# B&R Automation Studio project NAEUL004C00R13L518F00 (part 38)

#### Act_Alarm.st
```iecst
(** 2019-03-25 **)
ACTION Act_Alarm:

	//Error
	IF EDGEPOS(eStatus = Error) THEN

		tyAlmData.sProgNm		:= p_sProgNm;
		tyAlmData.udiCode		:= udiStatus;
		tyAlmData.eSeverity		:= AlmSeverityError;
		tyAlmData.udiRunTime	:= tyAlmData.udiRunTime + 1;
		tyAlmData.bAlm			:= TRUE;
		tyAlmData.udiModuleNum  := udiModuleNum;
		g_sUsrMgmtProgNm		:= p_sProgNm;

		//Get Error Message
		IF tyAlmData.udiCode < 10000 OR tyAlmData.udiCode > 10099 THEN
			tyAlmData.sAlmMsg	:= 'Unknown';
			tyAlmData.sRcyMsg	:= 'Unknown';
		ELSE
			tyAlmData.sAlmMsg	:= a_tyAlmText[tyAlmData.udiCode].sAlmText;
			tyAlmData.sRcyMsg	:= a_tyAlmText[tyAlmData.udiCode].sRcyText;
		END_IF

		sStatTxt	:= tyAlmData.sAlmMsg;

	ELSIF bRstErr AND (tyAlmData.udiCode <> 0) THEN

		tyAlmData.udiCode	:= 0;
		tyAlmData.eSeverity	:= AlmSeverityNA;
		tyAlmData.sAlmMsg	:= '';
		tyAlmData.sRcyMsg	:= '';
		tyAlmData.bAlm			:= FALSE;
		sStatTxt	:= a_sStatText[eStat];

	END_IF

END_ACTION
```

### Package Logical/OvenInfo - cmp

### OvenInfo.typ - Do Not Change!!!
```iecst
(*2018-12-13*)
(**)
(*Action*)

TYPE
	eOvenInfoAction :
		(
		OvenInfoActIdle,
		OvenInfoActSetBrdInOven,
		OvenInfoActSetOvenAllow,
		OvenInfoActRstOvenAllow
		);
	tyOvenInfo : 	STRUCT
		In : tyOvenInfoIn1;
		Out : tyOvenInfoOut1;
	END_STRUCT;
	tyOvenInfoIn1 : 	STRUCT
		eAct : eOvenInfoAction; (*Hardware Info's Action*)
		bPrep : BOOL := TRUE; (*Project Preparation*)
		bEn : BOOL := TRUE; (*Enable*)
		bDis : BOOL := FALSE; (*Disable*)
		bPrepExtdd : BOOL;
		bEnExtdd : BOOL;
		bDisExtdd : BOOL;
		bManual : BOOL;
		diBffrMtySlt : DINT;
		diAddBffr : DINT;
		diSetBrdInOven : DINT;
		bCntUp : BOOL;
		bCntDown : BOOL;
		bLinkOpsStatusRun : BOOL;
		eLinkOpsTravLifPosGo : REFERENCE TO eTravLifULPos;
		usiLinkProdRcpCurrRcpMcMod : REFERENCE TO USINT;
		diMinBffr : REFERENCE TO DINT;
		bBGRun : BOOL;
		BrdPerSlt : DINT;
		bLinkConvHvBrd : BOOL;
	END_STRUCT;
	tyOvenInfoOut1 : 	STRUCT
		eStat : eOvenInfoAction := OvenInfoActIdle; (*Hardware Info's State*)
		eStatus : eFBStatus := Idle; (*Hardware Info's Status*)
		sStatTxt : STRING[200] := ''; (*Hardware Info's State in Text*)
		tyAlmData : tyAlmDat; (*Alarm Data*)
		bOvenAllow : BOOL;
		diBrdInOven : DINT;
	END_STRUCT;
END_TYPE
```

### OvenInfo.var - Change By Project
```iecst
VAR
	g_tyOvenInfoA : tyOvenInfoOut1;
	g_tyOvenInfoB : tyOvenInfoOut1;
END_VAR
```

### Program Logical/OvenInfo/OvenInfoA (IEC, version 1.00.0) - 1.00.0 - NtOvenInfo v5.00.0

#### Init.st - Change By Project
```iecst
(** 2019-03-25 **)
PROGRAM _INIT

	(* Always Change If Project Change *)

	//Pass Address To Global Address For External Use
	//Action, State & Status
	p_OvenInfoAStat		:= ADR(eStat);
	p_OvenInfoAStatus	:= ADR(eStatus);
	p_OvenInfoAStatTxt	:= ADR(sStatTxt);

	//Alarm

	//Output
	p_OvenInfoAOvenAllow	:= ADR(bOvenAllow);
	p_OvenInfoABrdInOven	:= ADR(diBrdInOven);

	(* Always Change If Project Change *)

END_PROGRAM
```

#### Act_InitGlobal.st - Change By Project
```iecst
(** 2019-04-04 **)
ACTION Act_InitGlobal:

	(* Always Change If Project Change *)

	//Pass Data To Link
	p_bLinkOpsStatusRun ACCESS p_OpsStatusRun;
//	p_usiLinkProdRcpCurrRcpMcMod ACCESS p_ProdRcpCurrRcp2McMod;
	p_eLinkOpsTravLifPosGo ACCESS p_OpsTravLifULPosGo;
	p_eLinkConvStat ACCESS p_PshrConvStat;
	p_bLinkConvHvBrd ACCESS p_PshrConvHvBrd;

	//Pass Data To Internal Use
	p_eAct ACCESS p_UIOvenInfoAAct;
	p_bPrep ACCESS p_NtParamOvenInfoPrep;
	p_bEn ACCESS p_McParamOvenEn;
	p_bPrepExtdd ACCESS p_NtParamOvenInfoExtdPrep;
	p_bEnExtdd ACCESS p_McParamExtdOvenEn;
	p_bManual ACCESS p_UIMnlMod;
	p_diBffrMtySlt ACCESS p_BufferMagABffrMtySlt;
	//p_diMinBffr ACCESS p_ProdRcpCurrRcp2MinReqFreeBffr;
	p_diAddBffr ACCESS p_McParamOvenMaxBffr;
	p_diSetBrdInOven ACCESS p_UIOvenInfoSetBrdInOvenA;
	p_bCntUp ACCESS p_DIOvenInfeedSigA;
	p_bNtSettingsLoadDone ACCESS p_StartupNtSettingsLoadDone;

	p_bNtParamAutoRcpPrep ACCESS p_NtParamAutoRcpPrep;
	p_bMcParamAutoRcpDis  ACCESS p_McParamAutoRcpDisable;
	p_eNtParamAutoRcpPrecededBy ACCESS p_NtParamAutoRcpPrecededBy;
	(* Always Change If Project Change *)

END_ACTION
```

#### InputRef_Link.var - Change By Project
```iecst
(*2019-04-04*)
(**)
(*External*)
VAR
	p_bLinkOpsStatusRun : REFERENCE TO BOOL;
	p_usiLinkProdRcpCurrRcpMcMod : REFERENCE TO USINT;
	p_eLinkOpsTravLifPosGo : REFERENCE TO eTravLifULPos;
	p_eLinkConvStat : REFERENCE TO eConvAction;
	p_bLinkConvHvBrd : REFERENCE TO BOOL;
END_VAR
```

#### Act_LinkAction.st - Change By Project
```iecst
(** 2019-04-04 **)
ACTION Act_LinkAction:

	IF EDGENEG(p_bManual) THEN
		p_eAct	:= OvenInfoActIdle;
	END_IF

END_ACTION
```

#### Act_Link.st - Change By Project
```iecst
(** 2019-03-29 **)
ACTION Act_Link:
	IF g_tyNtParamCurr.bAutoRcpPrep AND NOT(g_tyMcParamCurr.bAutoRcpDisable) THEN //AutoRcp Ignored Follower
		tylocalOvenInfoA.In.usiLinkProdRcpCurrRcpMcMod ACCESS p_ProdRcpCurrRcp0McMod;
		tylocalOvenInfoA.In.diMinBffr ACCESS p_ProdRcpCurrRcp0MinReqFreeBffr;
	ELSE
		tylocalOvenInfoA.In.usiLinkProdRcpCurrRcpMcMod ACCESS p_ProdRcpCurrRcp1McMod;
		tylocalOvenInfoA.In.diMinBffr ACCESS p_ProdRcpCurrRcp2MinReqFreeBffr;
	END_IF

	tylocalOvenInfoA.In.bBGRun	:= tylocalOvenInfoA.In.bLinkOpsStatusRun
					AND (tylocalOvenInfoA.In.usiLinkProdRcpCurrRcpMcMod = ULModUnloadFrontLnA OR tylocalOvenInfoA.In.usiLinkProdRcpCurrRcpMcMod = ULModRejFrontLnA
					OR tylocalOvenInfoA.In.usiLinkProdRcpCurrRcpMcMod = ULModRejFrontLnARev OR tylocalOvenInfoA.In.usiLinkProdRcpCurrRcpMcMod = ULModUnloadDualLnAB
					OR tylocalOvenInfoA.In.usiLinkProdRcpCurrRcpMcMod = ULModRejDualLnA OR tylocalOvenInfoA.In.usiLinkProdRcpCurrRcpMcMod = ULModRejDualLnB);

	tylocalOvenInfoA.In.bCntDown 	:= tylocalOvenInfoA.In.eLinkOpsTravLifPosGo = TravLifULPosUS1 AND tylocalOvenInfoA.In.eLinkConvStat = ConvActEnt AND tylocalOvenInfoA.In.bLinkConvHvBrd = TRUE;

END_ACTION
```

#### Cyclic.st - Do Not Change!!!
```iecst
(** 2019-03-29 **)
PROGRAM _CYCLIC

	IF bInitialDone = FALSE THEN
		IF g_tyStartUp.bNtSettingsLoadDone = TRUE  THEN
			bInitialDone	:= TRUE;
			Act_Initial;
		END_IF

	ELSE

		IF (tylocalOvenInfoA.In.bPrep = TRUE) AND (tylocalOvenInfoA.In.bEn = TRUE) AND (tylocalOvenInfoA.In.bDis = FALSE) THEN
			Act_InputConfig;
			Act_Link;
			Act_Main;
			Act_OutputConfig;
		ELSE
			Act_Main_Disable;

			IF tylocalOvenInfoA.Out.eStat <> OvenInfoActIdle THEN
				tylocalOvenInfoA.Out.eStatus	:= Done;
			ELSE
				tylocalOvenInfoA.Out.eStatus	:= Idle;
			END_IF
		END_IF

	END_IF

END_PROGRAM
```

#### Act_Initial.st - Do Not Change!!!
```iecst
(** 2019-01-03 **)
ACTION Act_Initial:

	//Initial
	sStatTxt	:= a_sStatText[eStat];

	fbStd(bEn := FALSE);
	fbExtdd(bEn := FALSE);

END_ACTION
```

#### Act_Main.st - Do Not Change!!!
```iecst
(** 2019-01-10 **)
ACTION Act_Main:

	IF EDGENEG(g_tyUIOut.bManualMod) THEN
		tylocalOvenInfoA.In.eAct	:= OvenInfoActIdle;
	END_IF
	//Set tylocalOvenInfoA.In.eAct
	IF tylocalOvenInfoA.Out.eStatus = Idle OR tylocalOvenInfoA.Out.eStatus = Busy OR tylocalOvenInfoA.Out.eStatus = Done THEN
		tylocalOvenInfoA.Out.eStat	:= tylocalOvenInfoA.In.eAct;
	END_IF

	IF tylocalOvenInfoA.Out.eStatOld <> tylocalOvenInfoA.Out.eStat THEN
		tylocalOvenInfoA.Out.sStatTxt	:= a_sStatText[tylocalOvenInfoA.Out.eStat];

		tylocalOvenInfoA.Out.eStatOld	:= tylocalOvenInfoA.Out.eStat;

		tylocalOvenInfoA.Out.eStatus		:= Busy;
	END_IF

	//Main
	CASE tylocalOvenInfoA.Out.eStat OF

		OvenInfoActIdle:
			tylocalOvenInfoA.Out.eStatus	:= Idle;

		OvenInfoActSetBrdInOven:
			IF tylocalOvenInfoA.Out.eStatus = Idle OR tylocalOvenInfoA.Out.eStatus = Busy THEN

				tylocalOvenInfoA.Out.diBrdInOven	:= tylocalOvenInfoA.In.diSetBrdInOven;
				tylocalOvenInfoA.Out.eStatus		:= Done;

			END_IF

		OvenInfoActSetOvenAllow:
			IF tylocalOvenInfoA.Out.eStatus = Idle OR tylocalOvenInfoA.Out.eStatus = Busy THEN

				tylocalOvenInfoA.Out.bOvenAllow	:= TRUE;
				tylocalOvenInfoA.Out.eStatus		:= Done;

			END_IF

		OvenInfoActRstOvenAllow:
			IF tylocalOvenInfoA.Out.eStatus = Idle OR tylocalOvenInfoA.Out.eStatus = Busy THEN

				tylocalOvenInfoA.Out.bOvenAllow	:= FALSE;
				tylocalOvenInfoA.Out.eStatus		:= Done;

			END_IF

	END_CASE

	IF tylocalOvenInfoA.In.bManual = TRUE THEN
		fbStd(bEn := FALSE);
		fbExtdd(bEn := FALSE);

	ELSIF tylocalOvenInfoA.In.bBGRun = FALSE THEN
		fbStd(bEn := FALSE);
		fbExtdd(bEn := FALSE);

		tylocalOvenInfoA.Out.bOvenAllow	:= FALSE;

	ELSIF (tylocalOvenInfoA.In.bPrepExtdd = TRUE) AND (tylocalOvenInfoA.In.bEnExtdd = TRUE) AND (tylocalOvenInfoA.In.bDisExtdd = FALSE) THEN

		fbStd(bEn := FALSE);

		IF EDGEPOS(tylocalOvenInfoA.In.bCntUp) THEN
			tylocalOvenInfoA.Out.diBrdInOven	:= tylocalOvenInfoA.Out.diBrdInOven + 1;
		END_IF

		IF EDGEPOS(tylocalOvenInfoA.In.bCntDown) THEN
			tylocalOvenInfoA.Out.diBrdInOven	:= tylocalOvenInfoA.Out.diBrdInOven - 1;
		END_IF

		IF tylocalOvenInfoA.Out.diBrdInOven < 0 THEN
			tylocalOvenInfoA.Out.diBrdInOven	:= 0;
		END_IF

		fbExtdd.diAddBffr		:= tylocalOvenInfoA.In.diAddBffr;
		fbExtdd.diBffrMtySlt	:= tylocalOvenInfoA.In.diBffrMtySlt;
		fbExtdd.diBrdInOven		:= tylocalOvenInfoA.Out.diBrdInOven;
		fbExtdd.diBrdPerSlt		:= tylocalOvenInfoA.In.diBrdPerSlt;
		fbExtdd(bEn := TRUE);
		tylocalOvenInfoA.Out.bOvenAllow	:= fbExtdd.bOvenAllow;

	ELSE

		fbExtdd(bEn := FALSE);

		fbStd.diBffrMtySlt		:= tylocalOvenInfoA.In.diBffrMtySlt;
		fbStd.diMinBffrMtySlt	:= tylocalOvenInfoA.In.diMinBffr;
		fbStd(bEn := TRUE);
		tylocalOvenInfoA.Out.bOvenAllow	:= fbStd.bOvenAllow;

	END_IF

END_ACTION
```

#### Act_Main_Disable.st - Do Not Change!!!
```iecst
(** 2019-01-24 **)
ACTION Act_Main_Disable:

	tylocalOvenInfoA.Out.bOvenAllow	:= TRUE;

END_ACTION
```

#### InputRef.var - Do Not Change!!!
```iecst
(*2019-04-04*)
(**)
(*General*)
VAR
	p_eAct : REFERENCE TO eOvenInfoAction;
END_VAR
(**)
VAR
	p_bPrep : REFERENCE TO BOOL;
	p_bEn : REFERENCE TO BOOL;
	p_bDis : REFERENCE TO BOOL;
	p_bPrepExtdd : REFERENCE TO BOOL;
	p_bEnExtdd : REFERENCE TO BOOL;
	p_bDisExtdd : REFERENCE TO BOOL;
END_VAR
(**)
(*Configuration*)
VAR
	p_bBGRun : REFERENCE TO BOOL;
	p_bManual : REFERENCE TO BOOL;
	p_diBffrMtySlt : REFERENCE TO DINT;
	p_diMinBffr : REFERENCE TO DINT;
	p_diAddBffr : REFERENCE TO DINT;
	p_diBrdPerSlt : REFERENCE TO DINT;
	p_bCntUp : REFERENCE TO BOOL;
	p_bCntDown : REFERENCE TO BOOL;
	p_diSetBrdInOven : REFERENCE TO DINT;
	p_bNtSettingsLoadDone : REFERENCE TO BOOL;
END_VAR
(*AutoRcp*)
VAR
	p_bNtParamAutoRcpPrep : REFERENCE TO BOOL;
	p_bMcParamAutoRcpDis : REFERENCE TO BOOL;
	p_eNtParamAutoRcpPrecededBy : REFERENCE TO eAutoRcpPreceded;
END_VAR
```

#### Local.var - Do Not Change!!!
```iecst
(*2019-04-30*)
(**)
VAR
	tylocalOvenInfoA : tyOvenInfo;
	a_sStatText : ARRAY[0..50] OF STRING[200] := ['Idling','Setting Board In Oven Value','Turning On Oven Allow Output','Turning Off Oven Allow Output',47('')];
END_VAR
(**)
(*Local Alarm*)
(**)
(*Local Output*)
VAR
	bOvenAllow : BOOL;
END_VAR
VAR RETAIN
	diBrdInOven : DINT;
END_VAR
(**)
(*Local Input*)
VAR
	bPrep : BOOL := TRUE;
	bEn : BOOL := TRUE;
	bDis : BOOL := FALSE;
	bPrepExtdd : BOOL := TRUE;
	bEnExtdd : BOOL := TRUE;
	bDisExtdd : BOOL := FALSE;
	bBGRun : BOOL := FALSE;
	bManual : BOOL := FALSE;
	diBffrMtySlt : DINT;
	diMinBffr : DINT;
	diAddBffr : DINT;
	diBrdPerSlt : DINT := 1;
	bCntUp : BOOL;
	bCntDown : BOOL;
	diSetBrdInOven : DINT;
	bNtSettingsLoadDone : BOOL := TRUE;
END_VAR
(**)
(*Local*)
VAR
	bInitDone : BOOL;
	bInitialDone : BOOL;
	fbStd : fbOvenInfoStd;
	fbExtdd : fbOvenInfoExtdd;
	eStatOld : eOvenInfoAction := OvenInfoActIdle;
END_VAR
```

#### Act_InputConfig.st - not listed in the package file held
```iecst
ACTION Act_InputConfig:

	//Pass Data To Link
	tylocalOvenInfoA.In.bLinkOpsStatusRun :=  g_tyOps.bStatusRun;
	//	p_usiLinkProdRcpCurrRcpMcMod ACCESS p_ProdRcpCurrRcp2McMod;
	tylocalOvenInfoA.In.eLinkOpsTravLifPosGo ACCESS p_OpsTravLifULPosGo;
	tylocalOvenInfoA.In.eLinkConvStat := g_tyPshrConv.eStat;
	tylocalOvenInfoA.In.bLinkConvHvBrd := g_tyPshrConv.bHvBrd;

	//Pass Data To Internal Use
	tylocalOvenInfoA.In.eAct := g_tyUIOut.eOvenInfoAAct;
	tylocalOvenInfoA.In.bPrep := g_tyNtParam.bOvenInfoPrep;
	tylocalOvenInfoA.In.bEn := g_tyMcParamCurr.bOvenEn;
	tylocalOvenInfoA.In.bPrepExtdd := g_tyNtParam.bOvenInfoExtdPrep;
	tylocalOvenInfoA.In.bEnExtdd := g_tyMcParamCurr.bExtdOvenEn;
	tylocalOvenInfoA.In.bManual := g_tyUIOut.bMnlMod;
	tylocalOvenInfoA.In.diBffrMtySlt  := g_tyBufferMagA.diBffrMtySlt;
	//tylocalOvenInfoA.In.diMinBffr ACCESS p_ProdRcpCurrRcp2MinReqFreeBffr;
	tylocalOvenInfoA.In.diAddBffr := g_tyMcParamCurr.diOvenMaxBffr;
	tylocalOvenInfoA.In.diSetBrdInOven := g_tyUIOut.diOvenInfoSetBrdInOvenA;
	tylocalOvenInfoA.In.bCntUp := g_tyDInput.bOvenInfeedSigA;

	(* Always Change If Project Change *)

END_ACTION
```

#### Act_OutputConfig.st - not listed in the package file held
```iecst
ACTION Act_OutputConfig:

	g_tyOvenInfoA := tylocalOvenInfoA.Out;

END_ACTION
```

### Program Logical/OvenInfo/OvenInfoB (IEC) - 1.00.0 - NtOvenInfo v5.00.0

#### InputRef.var
```iecst
(*2019-04-04*)
(**)
(*General*)
VAR
	p_eAct : REFERENCE TO eOvenInfoAction;
END_VAR
(**)
VAR
	p_bPrep : REFERENCE TO BOOL;
	p_bEn : REFERENCE TO BOOL;
	p_bDis : REFERENCE TO BOOL;
	p_bPrepExtdd : REFERENCE TO BOOL;
	p_bEnExtdd : REFERENCE TO BOOL;
	p_bDisExtdd : REFERENCE TO BOOL;
END_VAR
(**)
(*Configuration*)
VAR
	p_bBGRun : REFERENCE TO BOOL;
	p_bManual : REFERENCE TO BOOL;
	p_diBffrMtySlt : REFERENCE TO DINT;
	p_diMinBffr : REFERENCE TO DINT;
	p_diAddBffr : REFERENCE TO DINT;
	p_diBrdPerSlt : REFERENCE TO DINT;
	p_bCntUp : REFERENCE TO BOOL;
	p_bCntDown : REFERENCE TO BOOL;
	p_diSetBrdInOven : REFERENCE TO DINT;
	p_bNtSettingsLoadDone : REFERENCE TO BOOL;
END_VAR
(*AutoRcp*)
VAR
	p_bNtParamAutoRcpPrep : REFERENCE TO BOOL;
	p_bMcParamAutoRcpDis1 : REFERENCE TO BOOL;
	p_eNtParamAutoRcpPrecededBy : REFERENCE TO eAutoRcpPreceded;
	p_bMcParamAutoRcpDis : REFERENCE TO BOOL;
END_VAR
```

#### InputRef_Link.var
```iecst
(*2019-04-04*)
(**)
(*External Data*)
VAR
	p_bLinkNtParamPrepB : REFERENCE TO BOOL;
	p_bLinkNtParamOvenInfoPrep : REFERENCE TO BOOL;
	p_bLinkOpsStatusRun : REFERENCE TO BOOL;
	p_usiLinkProdRcpCurrRcpMcMod : REFERENCE TO USINT;
	p_eLinkOpsTravLifPosGo : REFERENCE TO eTravLifULPos;
	p_eLinkConvStat : REFERENCE TO eConvAction;
	p_bLinkConvHvBrd : REFERENCE TO BOOL;
END_VAR
```

#### Local.var
```iecst
(*2019-04-30*)
VAR
	tylocalOvenInfoB : tyOvenInfo;
	a_sStatText : ARRAY[0..50] OF STRING[200] := ['Idling','Setting Board In Oven Value','Turning On Oven Allow Output','Turning Off Oven Allow Output',47('')];
END_VAR
(**)
(*Local Alarm*)
(**)
(*Local Output*)
VAR
	bOvenAllow : BOOL;
END_VAR
VAR RETAIN
	diBrdInOven : DINT;
END_VAR
(**)
(*Local Input*)
VAR
	bPrep : BOOL := TRUE;
	bEn : BOOL := TRUE;
	bDis : BOOL := FALSE;
	bPrepExtdd : BOOL := TRUE;
	bEnExtdd : BOOL := TRUE;
	bDisExtdd : BOOL := FALSE;
	bBGRun : BOOL := FALSE;
	bManual : BOOL := FALSE;
	diBffrMtySlt : DINT;
	diMinBffr : DINT;
	diAddBffr : DINT;
	diBrdPerSlt : DINT := 1;
	bCntUp : BOOL;
	bCntDown : BOOL;
	diSetBrdInOven : DINT;
	bNtSettingsLoadDone : BOOL := TRUE;
END_VAR
(**)
(*Local*)
VAR
	bInitDone : BOOL;
	bInitialDone : BOOL;
	fbStd : fbOvenInfoStd;
	fbExtdd : fbOvenInfoExtdd;
	eStatOld : eOvenInfoAction := OvenInfoActIdle;
END_VAR
```

#### Act_Background.st
```iecst
(** 2019-05-15 **)
ACTION Act_Background:

	IF p_bManual = TRUE THEN
		fbStd(bEn := FALSE);
		fbExtdd(bEn := FALSE);

	ELSIF p_bBGRun = FALSE THEN
		fbStd(bEn := FALSE);
		fbExtdd(bEn := FALSE);

		bOvenAllow	:= FALSE;

	ELSIF (p_bPrepExtdd = TRUE) AND (p_bEnExtdd = TRUE) AND (p_bDisExtdd = FALSE) THEN

		fbStd(bEn := FALSE);

		IF EDGEPOS(p_bCntUp) THEN
			diBrdInOven	:= diBrdInOven + 1;
		END_IF

		IF EDGEPOS(p_bCntDown) THEN
			diBrdInOven	:= diBrdInOven - 1;
		END_IF

		IF diBrdInOven < 0 THEN
			diBrdInOven	:= 0;
		END_IF

		fbExtdd.diAddBffr		:= p_diAddBffr;
		fbExtdd.diBffrMtySlt	:= p_diBffrMtySlt;
		fbExtdd.diBrdInOven		:= diBrdInOven;
		fbExtdd.diBrdPerSlt		:= p_diBrdPerSlt;
		fbExtdd(bEn := TRUE);
		bOvenAllow	:= fbExtdd.bOvenAllow;

	ELSE

		fbExtdd(bEn := FALSE);

		fbStd.diBffrMtySlt		:= p_diBffrMtySlt;
		fbStd.diMinBffrMtySlt	:= p_diMinBffr;
		fbStd(bEn := TRUE);
		bOvenAllow	:= fbStd.bOvenAllow;

	END_IF

END_ACTION
```

#### Act_InitGlobal.st
```iecst
(** 2019-04-04 **)
ACTION Act_InitGlobal:

	(* Always Change If Project Change *)

	//Pass Data To Link
	p_bLinkNtParamPrepB ACCESS p_NtParamProjLaneBPrep;
	p_bLinkNtParamOvenInfoPrep ACCESS p_NtParamOvenInfoPrep;
	p_bLinkOpsStatusRun ACCESS p_OpsStatusRun;
//	p_usiLinkProdRcpCurrRcpMcMod ACCESS p_ProdRcpCurrRcp2McMod;
	p_eLinkOpsTravLifPosGo ACCESS p_OpsTravLifULPosGo;
	p_eLinkConvStat ACCESS p_PshrConvStat;
	p_bLinkConvHvBrd ACCESS p_PshrConvHvBrd;

	//Pass Data To Internal Use
	p_eAct ACCESS p_UIOvenInfoBAct;
	p_bEn ACCESS p_McParamOvenEn;
	p_bPrepExtdd ACCESS p_NtParamOvenInfoExtdPrep;
	p_bEnExtdd ACCESS p_McParamExtdOvenEn;
	p_bManual ACCESS p_UIMnlMod;
	p_diBffrMtySlt ACCESS p_BufferMagBBffrMtySlt;
//	p_diMinBffr ACCESS p_ProdRcpCurrRcp2MinReqFreeBffr;
	p_diAddBffr ACCESS p_McParamOvenMaxBffr;
	p_diSetBrdInOven ACCESS p_UIOvenInfoSetBrdInOvenB;
	p_bCntUp ACCESS p_DIOvenInfeedSigB;
	p_bNtSettingsLoadDone ACCESS p_StartupNtSettingsLoadDone;

	p_bNtParamAutoRcpPrep ACCESS p_NtParamAutoRcpPrep;
	p_bMcParamAutoRcpDis  ACCESS p_McParamAutoRcpDisable;
	p_eNtParamAutoRcpPrecededBy ACCESS p_NtParamAutoRcpPrecededBy;
	(* Always Change If Project Change *)

END_ACTION
```

#### Act_Initial.st
```iecst
(** 2019-01-03 **)
ACTION Act_Initial:

	//Initial
	tylocalOvenInfoA.Out.sStatTxt	:= a_sStatText[tylocalOvenInfoA.Out.eStat];

	fbStd(bEn := FALSE);
	fbExtdd(bEn := FALSE);

END_ACTION
```

#### Act_InitLocal.st
```iecst
(** 2019-04-04 **)
ACTION Act_InitLocal:

	//Input Reference Link To Local Variable
	p_eAct ACCESS ADR(eAct);
	p_bPrep ACCESS ADR(bPrep);
	p_bEn ACCESS ADR(bEn);
	p_bDis ACCESS ADR(bDis);
	p_bPrepExtdd ACCESS ADR(bPrepExtdd);
	p_bEnExtdd ACCESS ADR(bEnExtdd);
	p_bDisExtdd ACCESS ADR(bDisExtdd);
	p_bBGRun ACCESS ADR(bBGRun);
	p_bManual ACCESS ADR(bManual);
	p_diMinBffr ACCESS ADR(diMinBffr);
	p_diAddBffr ACCESS ADR(diAddBffr);
	p_diBffrMtySlt ACCESS ADR(diBffrMtySlt);
	p_diBrdPerSlt ACCESS ADR(diBrdPerSlt);
	p_bCntUp ACCESS ADR(bCntUp);
	p_bCntDown ACCESS ADR(bCntDown);
	p_diSetBrdInOven ACCESS ADR(diSetBrdInOven);
	p_bNtSettingsLoadDone ACCESS ADR(bNtSettingsLoadDone);

END_ACTION
```

#### Act_InputConfig.st
```iecst
ACTION Act_InputConfig:

	(* Always Change If Project Change *)

	//Pass Data To Link
	tylocalOvenInfoB.In.bLinkOpsStatusRun :=  g_tyOps.bStatusRun;
	//	p_usiLinkProdRcpCurrRcpMcMod ACCESS p_ProdRcpCurrRcp2McMod;
	tylocalOvenInfoB.In.eLinkOpsTravLifPosGo ACCESS p_OpsTravLifULPosGo;
	tylocalOvenInfoB.In.eLinkConvStat := g_tyPshrConv.eStat;
	tylocalOvenInfoB.In.bLinkConvHvBrd := g_tyPshrConv.bHvBrd;

	tylocalOvenInfoB.In.eAct := g_tyUIOut.eOvenInfoBAct;
	//tylocalOvenInfoB.In.bPrep := g_tyNtParam.bOvenInfoPrep;
	tylocalOvenInfoB.In.bEn := g_tyMcParamCurr.bOvenEn;
	tylocalOvenInfoB.In.bPrepExtdd := g_tyNtParam.bOvenInfoExtdPrep;
	tylocalOvenInfoB.In.bEnExtdd := g_tyMcParamCurr.bExtdOvenEn;
	tylocalOvenInfoB.In.bManual := g_tyUIOut.bMnlMod;
	tylocalOvenInfoB.In.diBffrMtySlt  := g_tyBufferMagB.diBffrMtySlt;
	//tylocalOvenInfoB.In.diMinBffr ACCESS p_ProdRcpCurrRcp2MinReqFreeBffr;
	tylocalOvenInfoB.In.diAddBffr := g_tyMcParamCurr.diOvenMaxBffr;
	tylocalOvenInfoB.In.diSetBrdInOven := g_tyUIOut.diOvenInfoSetBrdInOvenB;
	tylocalOvenInfoB.In.bCntUp := g_tyDInput.bOvenInfeedSigB;

	//Link bPrep, bEn & bDis
	tylocalOvenInfoB.In.bPrep	:= g_tyNtParamCurr.bOvenInfoPrep AND g_tyNtParamCurr.bProjLaneBPrep;

END_ACTION
```

#### Act_Link.st
```iecst
(** 2019-03-29 **)
ACTION Act_Link:

	IF g_tyNtParamCurr.bAutoRcpPrep AND NOT(g_tyMcParamCurr.bAutoRcpDisable) THEN //AutoRcp Ignored Follower
		tylocalOvenInfoB.In.usiLinkProdRcpCurrRcpMcMod ACCESS p_ProdRcpCurrRcp0McMod;
		tylocalOvenInfoB.In.diMinBffr ACCESS p_ProdRcpCurrRcp0MinReqFreeBffr;
	ELSE
		tylocalOvenInfoB.In.usiLinkProdRcpCurrRcpMcMod ACCESS p_ProdRcpCurrRcp1McMod;
		tylocalOvenInfoB.In.diMinBffr ACCESS p_ProdRcpCurrRcp2MinReqFreeBffr;
	END_IF

	tylocalOvenInfoB.In.bBGRun := 	tylocalOvenInfoB.In.bLinkOpsStatusRun
					AND (tylocalOvenInfoB.In.usiLinkProdRcpCurrRcpMcMod = ULModUnloadRearLnB OR tylocalOvenInfoB.In.usiLinkProdRcpCurrRcpMcMod = ULModRejRearLnB
					OR tylocalOvenInfoB.In.usiLinkProdRcpCurrRcpMcMod = ULModRejRearLnBRev OR tylocalOvenInfoB.In.usiLinkProdRcpCurrRcpMcMod = ULModUnloadDualLnAB
					OR tylocalOvenInfoB.In.usiLinkProdRcpCurrRcpMcMod = ULModRejDualLnA OR tylocalOvenInfoB.In.usiLinkProdRcpCurrRcpMcMod = ULModRejDualLnB);

	tylocalOvenInfoA.In.bCntDown	:= p_eLinkOpsTravLifPosGo = TravLifULPosUS2 AND p_eLinkConvStat = ConvActEnt AND p_bLinkConvHvBrd = TRUE;

END_ACTION
```

#### Act_LinkEn.st
```iecst
(** 2019-01-11 **)
ACTION Act_LinkEn:

	//Link bPrep, bEn & bDis
	p_bPrep	:= p_bLinkNtParamOvenInfoPrep AND p_bLinkNtParamPrepB;

END_ACTION
```

#### Act_Main.st
```iecst
(** 2019-01-10 **)
ACTION Act_Main:

	IF EDGENEG(g_tyUIOut.bManualMod) THEN
		tylocalOvenInfoB.In.eAct	:= OvenInfoActIdle;
	END_IF
	//Set tylocalOvenInfoB.In.eAct
	IF tylocalOvenInfoB.Out.eStatus = Idle OR tylocalOvenInfoB.Out.eStatus = Busy OR tylocalOvenInfoB.Out.eStatus = Done THEN
		tylocalOvenInfoB.Out.eStat	:= tylocalOvenInfoB.In.eAct;
	END_IF

	IF tylocalOvenInfoB.Out.eStatOld <> tylocalOvenInfoB.Out.eStat THEN
		tylocalOvenInfoB.Out.sStatTxt	:= a_sStatText[tylocalOvenInfoB.Out.eStat];

		tylocalOvenInfoB.Out.eStatOld	:= tylocalOvenInfoB.Out.eStat;

		tylocalOvenInfoB.Out.eStatus		:= Busy;
	END_IF

	//Main
	CASE tylocalOvenInfoB.Out.eStat OF

		OvenInfoActIdle:
			tylocalOvenInfoB.Out.eStatus	:= Idle;

		OvenInfoActSetBrdInOven:
			IF tylocalOvenInfoB.Out.eStatus = Idle OR tylocalOvenInfoB.Out.eStatus = Busy THEN

				tylocalOvenInfoB.Out.diBrdInOven	:= tylocalOvenInfoB.In.diSetBrdInOven;
				tylocalOvenInfoB.Out.eStatus		:= Done;

			END_IF

		OvenInfoActSetOvenAllow:
			IF tylocalOvenInfoB.Out.eStatus = Idle OR tylocalOvenInfoB.Out.eStatus = Busy THEN

				tylocalOvenInfoB.Out.bOvenAllow	:= TRUE;
				tylocalOvenInfoB.Out.eStatus		:= Done;

			END_IF

		OvenInfoActRstOvenAllow:
			IF tylocalOvenInfoB.Out.eStatus = Idle OR tylocalOvenInfoB.Out.eStatus = Busy THEN

				tylocalOvenInfoB.Out.bOvenAllow	:= FALSE;
				tylocalOvenInfoB.Out.eStatus		:= Done;

			END_IF

	END_CASE

	IF tylocalOvenInfoB.In.bManual = TRUE THEN
		fbStd(bEn := FALSE);
		fbExtdd(bEn := FALSE);

	ELSIF tylocalOvenInfoB.In.bBGRun = FALSE THEN
		fbStd(bEn := FALSE);
		fbExtdd(bEn := FALSE);

		tylocalOvenInfoB.Out.bOvenAllow	:= FALSE;

	ELSIF (tylocalOvenInfoB.In.bPrepExtdd = TRUE) AND (tylocalOvenInfoB.In.bEnExtdd = TRUE) AND (tylocalOvenInfoB.In.bDisExtdd = FALSE) THEN

		fbStd(bEn := FALSE);

		IF EDGEPOS(tylocalOvenInfoB.In.bCntUp) THEN
			tylocalOvenInfoB.Out.diBrdInOven	:= tylocalOvenInfoB.Out.diBrdInOven + 1;
		END_IF

		IF EDGEPOS(tylocalOvenInfoB.In.bCntDown) THEN
			tylocalOvenInfoB.Out.diBrdInOven	:= tylocalOvenInfoB.Out.diBrdInOven - 1;
		END_IF

		IF tylocalOvenInfoB.Out.diBrdInOven < 0 THEN
			tylocalOvenInfoB.Out.diBrdInOven	:= 0;
		END_IF

		fbExtdd.diAddBffr		:= tylocalOvenInfoB.In.diAddBffr;
		fbExtdd.diBffrMtySlt	:= tylocalOvenInfoB.In.diBffrMtySlt;
		fbExtdd.Out.diBrdInOven		:= tylocalOvenInfoB.Out.diBrdInOven;
		fbExtdd.diBrdPerSlt		:= tylocalOvenInfoB.In.diBrdPerSlt;
		fbExtdd(bEn := TRUE);
		tylocalOvenInfoB.Out.bOvenAllow	:= fbExtdd.Out.bOvenAllow;

	ELSE

		fbExtdd(bEn := FALSE);

		fbStd.diBffrMtySlt		:= tylocalOvenInfoB.In.diBffrMtySlt;
		fbStd.diMinBffrMtySlt	:= tylocalOvenInfoB.In.diMinBffr;
		fbStd(bEn := TRUE);
		tylocalOvenInfoB.Out.bOvenAllow	:= fbStd.Out.bOvenAllow;

	END_IF

END_ACTION
```

#### Act_Main_Disable.st
```iecst
(** 2019-01-24 **)
ACTION Act_Main_Disable:

	tylocalOvenInfoB.Out.bOvenAllow= TRUE;

END_ACTION
```

#### Act_OutputConfig.st
```iecst
ACTION Act_OutputConfig:

	g_tyOvenInfoB := tylocalOvenInfoB.Out;

END_ACTION
```

#### Cyclic.st
```iecst
(** 2019-03-29 **)
PROGRAM _CYCLIC

	IF bInitialDone = FALSE THEN
		IF g_tyStartUp.bNtSettingsLoadDone = TRUE  THEN
			bInitialDone	:= TRUE;
			Act_Initial;
		END_IF

	ELSE

		IF (tylocalOvenInfoB.In.bPrep = TRUE) AND (tylocalOvenInfoB.In.bEn = TRUE) AND (tylocalOvenInfoB.In.bDis = FALSE) THEN
			Act_InputConfig;
			Act_Link;
			Act_Main;
			Act_OutputConfig;
		ELSE
			Act_Main_Disable;

			IF tylocalOvenInfoB.Out.eStat <> OvenInfoActIdle THEN
				tylocalOvenInfoB.Out.eStatus	:= Done;
			ELSE
				tylocalOvenInfoB.Out.eStatus	:= Idle;
			END_IF
		END_IF

	END_IF

END_PROGRAM
```

#### Init.st
```iecst
(** 2019-03-25 **)
PROGRAM _INIT

	(* Always Change If Project Change *)

	//Pass Address To Global Address For External Use
	//Action, State & Status
	p_OvenInfoBStat		:= ADR(eStat);
	p_OvenInfoBStatus	:= ADR(eStatus);
	p_OvenInfoBStatTxt	:= ADR(sStatTxt);

	//Alarm

	//Output
	p_OvenInfoBOvenAllow	:= ADR(bOvenAllow);
	p_OvenInfoBBrdInOven	:= ADR(diBrdInOven);

	(* Always Change If Project Change *)

END_PROGRAM
```

### OvenInfoA.var - not listed in the package file held
```iecst
(*2019-03-25*)
(**)
(*Action & State & Status*)
VAR
	p_OvenInfoAStat : UDINT;
	p_OvenInfoAStatus : UDINT;
	p_OvenInfoAStatTxt : UDINT;
END_VAR
(**)
(*Alarm*)
(**)
(*Output*)
VAR
	p_OvenInfoAOvenAllow : UDINT;
	p_OvenInfoABrdInOven : UDINT;
END_VAR
```

### OvenInfoB.var - not listed in the package file held
```iecst
(*2019-03-25*)
(**)
(*Action & State & Status*)
VAR
	p_OvenInfoBStat : UDINT;
	p_OvenInfoBStatus : UDINT;
	p_OvenInfoBStatTxt : UDINT;
END_VAR
(**)
(*Alarm*)
(**)
(*Output*)
VAR
	p_OvenInfoBOvenAllow : UDINT;
	p_OvenInfoBBrdInOven : UDINT;
END_VAR
```

### Buffer.typ - Do Not Change!!!
```iecst
(*2019-02-18*)
(**)
(*Action*)

TYPE
	eBufferAction :
		(
		BufferActIdle,
		BufferActCreateDir,
		BufferActGetRetainBffr,
		BufferActSetFull,
		BufferActSetMty,
		BufferActLoad,
		BufferActLoadSltChk,
		BufferActUnload,
		BufferActUnloadSltChk,
		BufferActUnloadCoolChk,
		BufferActUnloadSltChkCoolChk,
		BufferActNxtLoad,
		BufferActNxtLoadGd,
		BufferActNxtLoadBad,
		BufferActNxtUnload,
		BufferActNxtUnloadGd,
		BufferActNxtUnloadBad,
		BufferActChkCoolTm,
		BufferActChkCoolBrdAny,
		BufferActChkCoolBrdGd,
		BufferActChkCoolBrdBad,
		BufferActRstBffr,
		BufferActSetCoolFan,
		BufferActRstCoolFan,
		BufferActBGStartBffrSetFull,
		BufferActBGStartBffrSetMty,
		BufferActBGStopBffrSet,
		BufferActBGStartUpdtSen,
		BufferActBGStopUpdtSen,
		BufferActBGStartUpdtDisplay,
		BufferActBGStopUpdtDisplay,
		BufferActBGStartCoolFan,
		BufferActBGStopCoolFan
		);
	tyBuffer1 : 	STRUCT
		In : tyBufferIn1;
		Out : tyBufferOut1;
	END_STRUCT;
	tyBufferIn1 : 	STRUCT
		eAct : eBufferAction; (*Hardware Info's Action*)
		udiRstErr : UDINT;
		sFileName : STRING[80];
		bManual : BOOL;
		dtCurrDT : DATE_AND_TIME;
		diMinSlt : DINT;
		diMaxSlt : DINT;
		diPitch : DINT;
		diSltCap : DINT;
		diBffrTtlSlt : DINT;
		diCoolTm : DINT;
		diSltToSltInUM : DINT;
		diLifterBtmPosInUM : DINT;
		diLifterCurrPosInUM : DINT;
		bAscending : BOOL;
		bFIFO : BOOL;
		bGdBrdIn : BOOL;
		bGdBrdReq : BOOL;
		bNxtLoadSeq : BOOL;
		a_bSkip : ARRAY[1..c_diBffrSize]OF BOOL;
		diCoolFanOffDlyTm : DINT;
		bMagPresentSensor : BOOL;
		bPrepCoolFan : BOOL;
		bCoolFanTm : BOOL;
		tyBufferStat : tyBffrStat;
		sBffrNm : STRING[15];
		sProdNm : STRING[15];
		sBarcode1 : STRING[80];
		sBarcode2 : STRING[80];
		sCurrRcpNm : STRING[15];
		sProgNm : STRING[15];
		bNtSettingsLoadDone : BOOL;
		bNtParamAutoRcpPrep : BOOL;
		bMcParamAutoRcpDis : BOOL;
		bOpsMagConvULRlsMagAllw : BOOL;
		eNtParamCustomerReq : eCustomer;
		tyResponseFromMES : tyStatPlatformFromMES;
		diLinkSltToSltDist : REFERENCE TO DINT;
		bLinkMcParamProdSelTopToBtm : REFERENCE TO BOOL;
		bLinkPresentSen1 : BOOL;
		bLinkPresentSen2 : BOOL;
		bLinkOpsTravLifULExitBrd : REFERENCE TO BOOL;
	END_STRUCT;
	tyBufferOut1 : 	STRUCT
		eStat : eBufferAction := BufferActIdle; (*Hardware Info's State*)
		eStatus : eFBStatus := Idle; (*Hardware Info's Status*)
		sStatTxt : STRING[200] := ''; (*Hardware Info's State in Text*)
		tyAlmData : tyAlmDat; (*Alarm Data*)
		diNxtLoadSlt : DINT;
		diNxtUnloadSlt : DINT;
		diCoolBrdAny : DINT;
		diCoolBrdGd : DINT;
		diCoolBrdBad : DINT;
		bCoolNotRdy : BOOL;
		tyBuffer : tyBffr;
		tyDispBuffer : tyDispBffr;
		tyBufferStat : tyBffrStat;
		tyBoardUnloadStat : tyBrdUnloadStat;
		bCoolFanCtrl : BOOL;
		bParamDiff : BOOL;
		bMagRemoved : BOOL;
		bFIFOOld : BOOL;
		bMagPresent : BOOL;
		dtMagPresentTm : DATE_AND_TIME;
		diCurrSlt : DINT;
	END_STRUCT;
END_TYPE

(* *)

TYPE
	tyBufferMag : 	STRUCT
		In : tyBufferMagIn1;
		Out : tyBufferMagOut1;
	END_STRUCT;
	tyBufferMagIn1 : 	STRUCT
		eAct : eBufferAction; (*Hardware Info's Action*)
		udiRstErr : UDINT;
		bOpsStatusRun : BOOL;
		bBufferMagPresent1 : BOOL;
		bBufferMagPresent2 : BOOL;
		bBufferMagPresent3 : BOOL;
		bDIMagPresentSen1 : BOOL;
		bDIMagPresentSen2 : BOOL;
		bDIMagPresentSen3 : BOOL;
		tyBufferStat1 : tyBffrStat;
		tyBufferStat2 : tyBffrStat;
		tyBufferStat3 : tyBffrStat;
		bNtParamAutoRcpPrep : BOOL;
		bMcParamAutoRcpDis : BOOL;
		eNtParamMag : eULMag;
		bPrep : BOOL;
		bEn : BOOL;
		bDis : BOOL;
		usiProRcpProdSelMcMod : REFERENCE TO USINT;
	END_STRUCT;
	tyBufferMagOut1 : 	STRUCT
		eStat : eBufferAction := BufferActIdle; (*Hardware Info's State*)
		eStatus : eFBStatus := Idle; (*Hardware Info's Status*)
		sStatTxt : STRING[200] := ''; (*Hardware Info's State in Text*)
		tyAlmData : tyAlmDat; (*Alarm Data*)
		diBffrMtySlt : DINT;
	END_STRUCT;
END_TYPE
```

### Buffer.var - Change By Project
```iecst
VAR
	g_tyBuffer1 : tyBufferOut1;
	g_tyBuffer2 : tyBufferOut1;
	g_tyBuffer3 : tyBufferOut1;
	g_tyBufferMagA : tyBufferMagOut1;
	g_tyBufferMagB : tyBufferMagOut1;
END_VAR
```

### Program Logical/Buffer/Buffer1 (IEC) - 1.00.0 - NtBuffer v5.00.0 , NtFileIO v5.00.0

#### InputRef.var
```iecst
(*2019-07-03*)
(**)
(*General*)
VAR
	p_eAct : REFERENCE TO eBufferAction;
	p_udiRstErr : REFERENCE TO UDINT;
END_VAR
(**)
(*Configuration*)
VAR
	p_sFileName : REFERENCE TO STRING[80];
	p_bManual : REFERENCE TO BOOL;
	p_dtCurrDT : REFERENCE TO DATE_AND_TIME;
	p_diMinSlt : REFERENCE TO DINT;
	p_diMaxSlt : REFERENCE TO DINT;
	p_diPitch : REFERENCE TO DINT;
	p_diSltCap : REFERENCE TO DINT;
	p_diBffrTtlSlt : REFERENCE TO DINT;
	p_diCoolTm : REFERENCE TO DINT;
	p_diSltToSltInUM : REFERENCE TO DINT;
	p_diLifterBtmPosInUM : REFERENCE TO DINT;
	p_diLifterCurrPosInUM : REFERENCE TO DINT;
	p_bAscending : REFERENCE TO BOOL;
	p_bFIFO : REFERENCE TO BOOL;
	p_bGdBrdIn : REFERENCE TO BOOL;
	p_bGdBrdReq : REFERENCE TO BOOL;
	p_bNxtLoadSeq : REFERENCE TO BOOL;
	pa_bSkip : REFERENCE TO ARRAY[1..c_diBffrSize] OF BOOL;
	p_diCoolFanOffDlyTm : REFERENCE TO DINT;
	p_bMagPresentSensor : REFERENCE TO BOOL;
	p_bPrepCoolFan : REFERENCE TO BOOL;
	p_bCoolFanTm : REFERENCE TO BOOL;
	p_tyBuffer : REFERENCE TO tyBffr;
	p_tyDispBuffer : REFERENCE TO tyDispBffr;
	p_tyBufferStat : REFERENCE TO tyBffrStat;
	p_sBffrNm : REFERENCE TO STRING[15];
	p_sProdNm : REFERENCE TO STRING[15];
	p_sBarcode1 : REFERENCE TO STRING[80];
	p_sBarcode2 : REFERENCE TO STRING[80];
	p_sCurrRcpNm : REFERENCE TO STRING[15];
	p_sProgNm : REFERENCE TO STRING[15];
	p_bNtSettingsLoadDone : REFERENCE TO BOOL;
	p_bNtParamAutoRcpPrep : REFERENCE TO BOOL;
	p_bMcParamAutoRcpDis : REFERENCE TO BOOL;
	p_bOpsMagConvULRlsMagAllw : REFERENCE TO BOOL;
	p_eNtParamCustomerReq : REFERENCE TO eCustomer;
	p_tyResponseFromMES : REFERENCE TO tyStatPlatformFromMES;
	p_bNtParamAutoRcpF1ArbitraryType : REFERENCE TO BOOL;
END_VAR
```

#### InputRef_Link.var
```iecst
(*2019-04-09*)
(**)
(*External*)
VAR
	p_bLinkStartupRun : REFERENCE TO BOOL;
	p_bLinkNtParamProjMagConvPrep : REFERENCE TO BOOL;
	p_eLinkOpsMagULBufferAct : REFERENCE TO eBufferAction;
	p_eLinkOpsMagConvULBufferAct : REFERENCE TO eBufferAction;
	p_eLinkUIBufferAct : REFERENCE TO eBufferAction;
	p_bLinkOpsMagStepBffrLoad : REFERENCE TO BOOL;
END_VAR
(**)
VAR
	p_diLinkSltToSltDist : REFERENCE TO DINT;
	p_bLinkMcParamProdSelTopToBtm : REFERENCE TO BOOL;
	p_bLinkPresentSen1 : REFERENCE TO BOOL;
	p_bLinkPresentSen2 : REFERENCE TO BOOL;
	p_bLinkProjLifterMagPlatform : REFERENCE TO BOOL;
	p_eLinkOpsLifMagULBufferAct : REFERENCE TO eBufferAction;
	p_bLinkOpsTravLifULExitBrd : REFERENCE TO BOOL;
END_VAR
```

#### Local.var
```iecst
(*2019-06-07*)
(**)
(*Local Action, State & Status*)
VAR
	tylocalBuffer : tyBuffer1;
	eAct : eBufferAction;
	udiStatus : UDINT := 0;
	a_sStatText : ARRAY[0..50] OF STRING[200] := ['Idling','Creating Directory','Getting Retained Buffer Data','Setting Buffer Full','Setting Buffer Empty','Loading Board','Loading Board With Slot Check','Unloading Board','Unloading Board With Slot Check','Unloading Board With Cooling Time Check','Unloading Board With Slot Check And Cooling Time Check','Getting Next Load Board Slot Number','Getting Next Load Good Board Slot Number','Getting Next Load Bad Board Slot Number','Getting Next Unload Board Slot Number','Getting Next Unload Good Board Slot Number','Getting Next Unload Bad Board Slot Number','Checking Cooling Time','Checking Cooling Board','Checking Cooling Good Board','Checking Cooling Bad Board','Resetting Buffer','Turning On Cooling Fan','Turning Off Cooling Fan','Background Starting Buffer Set Full','Background Starting Buffer Set Empty','Background Stopping Buffer Set','Background Starting Update Sensor','Background Stopping Update Sensor','Background Starting Update Display','Background Stopping Update Display','Background Starting Cooling Fan','Background Stopping Cooling Fan',18('')];
END_VAR
(**)
(*Local Alarm*)
VAR
	tyAlmData : tyAlmDat;
	a_tyAlmText : ARRAY[10000..10099] OF tyAlmTxt := [(sAlmText:='Create User Directory Error',sRcyText:='An Error Occurred While Attempting To Create User Directory. Please Contact Nutek For A Possible Solution'),(sAlmText:='Create Retain Directory Error',sRcyText:='An Error Occurred While Attempting To Create Retain Directory. Please Contact Nutek For A Possible Solution'),(sAlmText:='File Open Error While Reading Retain File',sRcyText:='An Error Was Encountered While Trying To Open File. Please Contact Nutek For A Possible Solution.'),(sAlmText:='File Read Error While Reading Retain File',sRcyText:='An Error Was Encountered While Trying To Read File. Please Contact Nutek For A Possible Solution.'),(sAlmText:='File Close Error While Reading Retain File',sRcyText:='An Error Was Encountered While Trying To Close File. Please Contact Nutek For A Possible Solution.'),(sAlmText:='File Open Error While Setting Full Buffer',sRcyText:='An Error Was Encountered While Trying To Open File. Please Contact Nutek For A Possible Solution.'),(sAlmText:='File Create Error While Setting Full Buffer',sRcyText:='An Error Was Encountered While Trying To Create File. Please Contact Nutek For A Possible Solution.'),(sAlmText:='File Write Error While Setting Full Buffer',sRcyText:='An Error Was Encountered While Trying To Write File. Please Contact Nutek For A Possible Solution.'),(sAlmText:='File Close Error While Setting Full Buffer',sRcyText:='An Error Was Encountered While Trying To Close File. Please Contact Nutek For A Possible Solution.'),(sAlmText:='File Open Error While Setting Empty Buffer',sRcyText:='An Error Was Encountered While Trying To Open File. Please Contact Nutek For A Possible Solution.'),(sAlmText:='File Create Error While Setting Empty Buffer',sRcyText:='An Error Was Encountered While Trying To Create File. Please Contact Nutek For A Possible Solution.'),(sAlmText:='File Write Error While Setting Empty Buffer',sRcyText:='An Error Was Encountered While Trying To Write File. Please Contact Nutek For A Possible Solution.'),(sAlmText:='File Close Error While Setting Empty Buffer',sRcyText:='An Error Was Encountered While Trying To Close File. Please Contact Nutek For A Possible Solution.'),(sAlmText:='File Open Error While Loading Info To Buffer',sRcyText:='An Error Was Encountered While Trying To Open File. Please Contact Nutek For A Possible Solution.'),(sAlmText:='File Create Error While Loading Info To Buffer',sRcyText:='An Error Was Encountered While Trying To Create File. Please Contact Nutek For A Possible Solution.'),(sAlmText:='File Write Error While Loading Info To Buffer',sRcyText:='An Error Was Encountered While Trying To Write File. Please Contact Nutek For A Possible Solution.'),(sAlmText:='File Close Error While Loading Info To Buffer',sRcyText:='An Error Was Encountered While Trying To Close File. Please Contact Nutek For A Possible Solution.'),(sAlmText:='Wrong Slot Number To Load',sRcyText:='Invalid Slot to Load The Board.'),(sAlmText:='File Open Error While Loading Info To Buffer With Slot Check',sRcyText:='An Error Was Encountered While Trying To Open File. Please Contact Nutek For A Possible Solution.'),(sAlmText:='File Create Error While Loading Info To Buffer With Slot Check',sRcyText:='An Error Was Encountered While Trying To Create File. Please Contact Nutek For A Possible Solution.'),(sAlmText:='File Write Error While Loading Info To Buffer With Slot Check',sRcyText:='An Error Was Encountered While Trying To Write File. Please Contact Nutek For A Possible Solution.'),(sAlmText:='File Close Error While Loading Info To Buffer With Slot Check',sRcyText:='An Error Was Encountered While Trying To Close File. Please Contact Nutek For A Possible Solution.'),(sAlmText:='File Open Error While Unloading Info From Buffer',sRcyText:='An Error Was Encountered While Trying To Open File. Please Contact Nutek For A Possible Solution.'),(sAlmText:='File Create Error While Unloading Info From Buffer',sRcyText:='An Error Was Encountered While Trying To Create File. Please Contact Nutek For A Possible Solution.'),(sAlmText:='File Write Error While Unloading Info From Buffer',sRcyText:='An Error Was Encountered While Trying To Write File. Please Contact Nutek For A Possible Solution.'),(sAlmText:='File Close Error While Unloading Info From Buffer',sRcyText:='An Error Was Encountered While Trying To Close File. Please Contact Nutek For A Possible Solution.'),(sAlmText:='Wrong Slot Number To Unload',sRcyText:='Invalid Slot to Unload The Board.'),(sAlmText:='File Open Error While Unloading Info From Buffer With Slot Check',sRcyText:='An Error Was Encountered While Trying To Open File. Please Contact Nutek For A Possible Solution.'),(sAlmText:='File Create Error While Unloading Info From Buffer With Slot Check',sRcyText:='An Error Was Encountered While Trying To Create File. Please Contact Nutek For A Possible Solution.'),(sAlmText:='File Write Error While Unloading Info From Buffer With Slot Check',sRcyText:='An Error Was Encountered While Trying To Write File. Please Contact Nutek For A Possible Solution.'),(sAlmText:='File Close Error While Unloading Info From Buffer With Slot Check',sRcyText:='An Error Was Encountered While Trying To Close File. Please Contact Nutek For A Possible Solution.'),(sAlmText:='File Open Error While Unloading Info From Buffer With Cooling Time Check',sRcyText:='An Error Was Encountered While Trying To Open File. Please Contact Nutek For A Possible Solution.'),(sAlmText:='File Create Error While Unloading Info From Buffer With Cooling Time Check',sRcyText:='An Error Was Encountered While Trying To Create File. Please Contact Nutek For A Possible Solution.'),(sAlmText:='File Write Error While Unloading Info From Buffer With Cooling Time Check',sRcyText:='An Error Was Encountered While Trying To Write File. Please Contact Nutek For A Possible Solution.'),(sAlmText:='File Close Error While Unloading Info From Buffer With Cooling Time Check',sRcyText:='An Error Was Encountered While Trying To Close File. Please Contact Nutek For A Possible Solution.'),(sAlmText:='Wrong Slot Number To Unload With Cooling Time Check',sRcyText:='Invalid Slot to Unload The Board with Cooling Time Check.'),(sAlmText:='File Open Error While Unloading Info From Buffer With Slot Check And Cooling Time Check',sRcyText:='An Error Was Encountered While Trying To Open File. Please Contact Nutek For A Possible Solution.'),(sAlmText:='File Create Error While Unloading Info From Buffer With Slot Check And Cooling Time Check',sRcyText:='An Error Was Encountered While Trying To Create File. Please Contact Nutek For A Possible Solution.'),(sAlmText:='File Write Error While Unloading Info From Buffer With Slot Check And Cooling Time Check',sRcyText:='An Error Was Encountered While Trying To Write File. Please Contact Nutek For A Possible Solution.'),(sAlmText:='File Close Error While Unloading Info From Buffer With Slot Check And Cooling Time Check',sRcyText:='An Error Was Encountered While Trying To Close File. Please Contact Nutek For A Possible Solution.'),(sAlmText:='Directory Does Not Exist While Setting Full Buffer',sRcyText:='The Directory Does Not Exist. Please Contact Nutek For A Possible Solution.'),(sAlmText:='Directory Does Not Exist While Setting Empty Buffer',sRcyText:='The Directory Does Not Exist. Please Contact Nutek For A Possible Solution.'),(sAlmText:='Directory Does Not Exist While Loading Info To Buffer',sRcyText:='The Directory Does Not Exist. Please Contact Nutek For A Possible Solution.'),(sAlmText:='Directory Does Not Exist While Loading Info To Buffer With Slot Check',sRcyText:='The Directory Does Not Exist. Please Contact Nutek For A Possible Solution.'),(sAlmText:='Directory Does Not Exist While Unloading Info From Buffer',sRcyText:='The Directory Does Not Exist. Please Contact Nutek For A Possible Solution.'),(sAlmText:='Directory Does Not Exist While Unloading Info From Buffer With Slot Check',sRcyText:='The Directory Does Not Exist. Please Contact Nutek For A Possible Solution.'),(sAlmText:='Directory Does Not Exist While Unloading Info From Buffer With Cooling Time Check',sRcyText:='The Directory Does Not Exist. Please Contact Nutek For A Possible Solution.'),(sAlmText:='Directory Does Not Exist While Unloading Info From Buffer With Slot Check And Cooling Time Check',sRcyText:='The Directory Does Not Exist. Please Contact Nutek For A Possible Solution.'),(sAlmText:='Unloading Slot Is Skipped While Unloading Buffer',sRcyText:='Unload From Wrong Slot (Skip Slot).'),(sAlmText:='Unloading Slot Is Not For Board While Unloading Buffer',sRcyText:='Unload From Wrong Slot (Not For Board).'),(sAlmText:='Unloading Slot Board Is Not Available While Unloading Buffer',sRcyText:='Unload From Wrong Slot (Board Is Not Available).'),(sAlmText:='Unloading Last Sub Slot Is Not For Board While Unloading Buffer',sRcyText:='Unload From Wrong Slot (Last Sub Slot Is Not For Board).'),(sAlmText:='Unloading Last Sub Slot Has No Board While Unloading Buffer',sRcyText:='Unload From Wrong Slot (Last Sub Slot Has No Board).'),(sAlmText:='Board Quantity In Slot Is 0 While Unloading Buffer',sRcyText:='Unload From Wrong Slot (Board Quantity In Slot = 0).'),(sAlmText:='Board Capacity In Slot Is 0 While Unloading Buffer',sRcyText:='Unload From Wrong Slot (Board Capacity In Slot = 0).'),(sAlmText:='Unloading Slot Is Skipped While Unloading Buffer With Slot Check',sRcyText:='Unload From Wrong Slot (Skip Slot).'),(sAlmText:='Unloading Slot Is Not For Board While Unloading Buffer With Slot Check',sRcyText:='Unload From Wrong Slot (Not For Board).'),(sAlmText:='Unloading Slot Board Is Not available While Unloading Buffer With Slot Check',sRcyText:='Unload From Wrong Slot (Board Is Not Available).'),(sAlmText:='Unloading Last Sub Slot Is Not For Board While Unloading Buffer With Slot Check',sRcyText:='Unload From Wrong Slot (Last Sub Slot Is Not For Board).'),(sAlmText:='Unloading Last Sub Slot Has No Board While Unloading Buffer With Slot Check',sRcyText:='Unload From Wrong Slot (Last Sub Slot Has No Board).'),(sAlmText:='Board Quantity In Slot Is 0 While Unloading Buffer With Slot Check',sRcyText:='Unload From Wrong Slot (Board Quantity In Slot = 0).'),(sAlmText:='Board Capacity In Slot Is 0 While Unloading Buffer With Slot Check',sRcyText:='Unload From Wrong Slot (Board Capacity In Slot = 0).'),(sAlmText:='Unloading Slot Is Skipped While Unloading Buffer With Cool Check',sRcyText:='Unload From Wrong Slot (Skip Slot).'),(sAlmText:='Unloading Slot Is Not For Board While Unloading Buffer With Cool Check',sRcyText:='Unload From Wrong Slot (Not For Board).'),(sAlmText:='Unloading Slot Board Is Not available While Unloading Buffer With Cool Check',sRcyText:='Unload From Wrong Slot (Board Is Not Available).'),(sAlmText:='Unloading Last Sub Slot Is Not For Board While Unloading Buffer With Cool Check',sRcyText:='Unload From Wrong Slot (Last Sub Slot Is Not For Board).'),(sAlmText:='Unloading Last Sub Slot Has No Board While Unloading Buffer With Cool Check',sRcyText:='Unload From Wrong Slot (Last Sub Slot Has No Board).'),(sAlmText:='Board Quantity In Slot Is 0 While Unloading Buffer With Cool Check',sRcyText:='Unload From Wrong Slot (Board Quantity In Slot = 0).'),(sAlmText:='Board Capacity In Slot Is 0 While Unloading Buffer With Cool Check',sRcyText:='Unload From Wrong Slot (Board Capacity In Slot = 0).'),(sAlmText:='Unloading Slot Is Skipped While Unloading Buffer With Cool & Slot Check',sRcyText:='Unload From Wrong Slot (Skip Slot).'),(sAlmText:='Unloading Slot Is Not For Board While Unloading Buffer With Cool & Slot Check',sRcyText:='Unload From Wrong Slot (Not For Board).'),(sAlmText:='Unloading Slot Board Is Not available While Unloading Buffer With Cool & Slot Check',sRcyText:='Unload From Wrong Slot (Board Is Not Available).'),(sAlmText:='Unloading Last Sub Slot Is Not For Board While Unloading Buffer With Cool & Slot Check',sRcyText:='Unload From Wrong Slot (Last Sub Slot Is Not For Board).'),(sAlmText:='Unloading Last Sub Slot Has No Board While Unloading Buffer With Cool & Slot Check',sRcyText:='Unload From Wrong Slot (Last Sub Slot Has No Board).'),(sAlmText:='Board Quantity In Slot Is 0 While Unloading Buffer With Cool & Slot Check',sRcyText:='Unload From Wrong Slot (Board Quantity In Slot = 0).'),(sAlmText:='Board Capacity In Slot Is 0 While Unloading Buffer With Cool & Slot Check',sRcyText:='Unload From Wrong Slot (Board Capacity In Slot = 0).'),(sAlmText:='Loading Slot Is Not For Board',sRcyText:='Load To Wrong Slot (Not For Board).'),(sAlmText:='Loading Slot Is Full Of Board',sRcyText:='Load To Wrong Slot (Full With Board).'),(sAlmText:='Loading First Sub-Slot Is Not For Board',sRcyText:='Load To Wrong Slot (First Sub Slot Not For Board).'),(sAlmText:='Loading Last Sub-Slot Have Board, Which Mean Slot Is Full Of Board',sRcyText:='Load To Wrong Slot (Full With Board(Last Sub Slot Have Board)).'),(sAlmText:='Loading Last Sub-Slot Is Not For Board',sRcyText:='Load To Wrong Slot (Last Sub Slot Not For Board).'),(sAlmText:='Loading Slot Is Full Of Board',sRcyText:='Load To Wrong Slot (Full With Board).'),(sAlmText:='Loading Slot Is Skipped',sRcyText:='Load To Wrong Slot (Skip Slot).'),(sAlmText:='Existing Board Status Is Different With Loading Board Status',sRcyText:='Existing Board Status Is Different With Loading Buffer Status.'),(sAlmText:='Loading Slot Is Not For Board',sRcyText:='Load To Wrong Slot (Not For Board).'),(sAlmText:='Loading Slot Is Full Of Board',sRcyText:='Load To Wrong Slot (Full With Board).'),(sAlmText:='Loading First Sub-Slot Is Not For Board',sRcyText:='Load To Wrong Slot (First Sub Slot Not For Board).'),(sAlmText:='Loading Last Sub-Slot Have Board, Which Mean Slot Is Full Of Board',sRcyText:='Load To Wrong Slot (Full With Board(Last Sub Slot Have Board)).'),(sAlmText:='Loading Last Sub-Slot Is Not For Board',sRcyText:='Load To Wrong Slot (Last Sub Slot Not For Board).'),(sAlmText:='Loading Slot Is Full Of Board',sRcyText:='Load To Wrong Slot (Full With Board).'),(sAlmText:='Loading Slot Is Skipped',sRcyText:='Load To Wrong Slot (Skip Slot).'),(sAlmText:='Existing Board Status Is Different With Loading Board Status',sRcyText:='Existing Board Status Is Different With Loading Buffer Status.'),8((0))];
END_VAR
(**)
(**)
(**)
(*Local*)
VAR
	bRstErr : BOOL;
	udiRstErrOld : UDINT;
	bInitDone : BOOL;
	bInitialDone : BOOL;
	bUpdateSensor : BOOL;
	bBffrSetMty : BOOL;
	bBffrSetFull : BOOL;
	bUpdtDisplay : BOOL;
	usiStep : USINT;
	diCurrSlt : DINT;
	diExpectedSlt : DINT;
	bSetFull : BOOL;
	bSetMty : BOOL;
	bCoolFanRun : BOOL;
	tyBffrParameter : tyBffrParam;
	fbDirCreate1 : fbDirCreate;
	fbDirCreate2 : fbDirCreate;
	fbFileRead1 : fbFileFullRead;
	fbFileWrite1 : fbFileFullWrite;
	fbCoolFanOffDlyTm : TON;
	fbCoolFanOffChkTm : TON := (PT:=T#500ms);
	fbMagAbsentTm : TON := (PT:=T#5s);
	fbMagPresentTm : TON := (PT:=T#8s);
	eStatOld : eBufferAction := BufferActIdle;
	bMESTrigSetFull : BOOL;
	bFileNotFound : BOOL;
	bNewProduct : BOOL;
	bLastProductUnload : BOOL;
	bLastProductLeftInBffr : BOOL;
	udiModuleNum : UDINT := 2001;
END_VAR
```

#### Act_Background.st
```iecst
(** 2019-07-03 **)
ACTION Act_Background:

	fbMagPresentTm(IN := p_bMagPresentSensor);

	//Update Retain
	IF bUpdateSensor = TRUE THEN
		bMagPresent	:= fbMagPresentTm.Q;
	END_IF

	//Display Buffer
	IF bUpdtDisplay = TRUE THEN
		fDispBffrDescending(ADR(p_tyDispBuffer) , tyBffrParameter , p_tyBuffer , p_dtCurrDT , DINT_TO_TIME(p_diCoolTm) , 0 , 1 , 2);
	END_IF

	//Cooling Fan Control
	IF p_bManual = TRUE THEN
		;

	ELSIF bCoolFanRun = TRUE AND p_bPrepCoolFan = TRUE AND bCoolFanTm = TRUE THEN //Cooling Fan Control By Cooling Time

		fbCoolFanOffChkTm(IN := TRUE);

		IF fbCoolFanOffChkTm.Q = TRUE THEN
			IF fBffrChkCoolBrdAny(p_dtCurrDT, DINT_TO_TIME(p_diCoolTm), p_tyBuffer) = 0 THEN
				fbCoolFanOffDlyTm.IN	:= TRUE;
			ELSE
				fbCoolFanOffDlyTm.IN	:= FALSE;
				bCoolFanCtrl			:= TRUE;
			END_IF

			fbCoolFanOffChkTm(IN := FALSE);
		END_IF

		fbCoolFanOffDlyTm;

		IF fbCoolFanOffDlyTm.Q = TRUE THEN
			bCoolFanCtrl	:= FALSE;
		END_IF

	ELSIF bCoolFanRun = TRUE AND p_bPrepCoolFan = TRUE AND bCoolFanTm = FALSE THEN	//Cooling Fan Control By Buffer Empty
		fbCoolFanOffDlyTm(IN := p_tyBufferStat.bBffrMty);

		IF p_tyBufferStat.bBffrMty = FALSE THEN
			bCoolFanCtrl	:= TRUE;
		END_IF

		IF fbCoolFanOffDlyTm.Q = TRUE THEN
			bCoolFanCtrl	:= FALSE;
		END_IF

	ELSE

		bCoolFanCtrl	:= FALSE;

	END_IF

	//Set Buffer By Magazine Present
	IF bBffrSetFull = TRUE THEN
		IF p_bMagPresentSensor = TRUE AND fbMagAbsentTm.Q = TRUE THEN
			bSetFull		:= TRUE;
			dtMagPresentTm	:= p_dtCurrDT;
		END_IF

		IF bSetFull = TRUE  THEN
			p_eAct	:= BufferActSetFull;

			IF eStatus = Done AND eStat = BufferActSetFull THEN
				p_eAct		:= BufferActIdle;
				bSetFull	:= FALSE;
			ELSIF eStatus = Error THEN
				bSetFull	:= FALSE;
			END_IF
		END_IF

		fbMagAbsentTm(IN := NOT p_bMagPresentSensor);

	ELSIF bBffrSetMty = TRUE THEN
		IF p_bMagPresentSensor = TRUE AND fbMagAbsentTm.Q = TRUE THEN
			bSetMty			:= TRUE;
			dtMagPresentTm	:= p_dtCurrDT;
		END_IF

		IF bSetMty = TRUE  THEN
			p_eAct	:= BufferActSetMty;

			IF eStatus = Done AND eStat = BufferActSetMty THEN
				p_eAct	:= BufferActIdle;
				bSetMty	:= FALSE;
			ELSIF eStatus = Error THEN
				bSetMty	:= FALSE;
			END_IF
		END_IF

		fbMagAbsentTm(IN := NOT p_bMagPresentSensor);

	END_IF

	//Check Parameter Different
	bParamDiff	:= (tyBffrParameter.bAscending <> p_bAscending)
	OR (tyBffrParameter.diMinSlt <> p_diMinSlt)
	OR (tyBffrParameter.diMaxSlt <> p_diMaxSlt)
	OR (tyBffrParameter.diPitch <> p_diPitch)
	OR (tyBffrParameter.diSltCap <> p_diSltCap)
	OR (bFIFOOld <> p_bFIFO);

	//Update MagRemoved
	bMagRemoved	:= fbMagAbsentTm.Q;

END_ACTION
```

#### Act_InitGlobal.st
```iecst
(** 2019-04-26 **)
ACTION Act_InitGlobal:

	(* Always Change If Project Change *)

	//Pass Data To Link
	p_bLinkStartupRun ACCESS p_StartupRun;
	p_bLinkNtParamProjMagConvPrep ACCESS p_NtParamProjMag1ConvPrep;
//	p_eLinkOpsMagULBufferAct ACCESS p_OpsMagUL1BufferAct;
	p_eLinkOpsMagConvULBufferAct ACCESS p_OpsMagConvUL1BufferAct;
	p_eLinkUIBufferAct ACCESS p_UIBuffer1Act;
	p_bLinkOpsMagStepBffrLoad ACCESS p_OpsMagConvUL1StepBffrLoad;
	p_bLinkProjLifterMagPlatform ACCESS p_NtParamProjLifterMagPlatform;
	p_eLinkOpsLifMagULBufferAct ACCESS p_OpsLifMagULBufferAct1;

	p_diLinkSltToSltDist ACCESS p_MagRcpCurrRcpSltToSlt;
	p_bLinkMcParamProdSelTopToBtm ACCESS p_ProdRcpCurrRcp2TopToBtm;
	p_bLinkPresentSen1 ACCESS p_DIMagPresentSen1;
	p_bLinkPresentSen2 ACCESS p_DIMagConvEntSen1;
	p_bLinkOpsTravLifULExitBrd ACCESS p_OpsTravLifULExitBrd;

	//Pass Data To Internal Use
	p_udiRstErr ACCESS p_RstErrReset;
	p_sFileName ACCESS p_NtParamBffr1FileNm;
	p_bManual ACCESS p_UIMnlMod;
	p_dtCurrDT ACCESS p_TimeCurrDT;
//	p_diMinSlt ACCESS p_ProdRcpCurrRcp2MinSltValue;
//	p_diMaxSlt ACCESS p_ProdRcpCurrRcp2MaxSltValue;
//	p_diPitch ACCESS p_ProdRcpCurrRcp2Pitch;
	p_diBffrTtlSlt ACCESS p_MagRcpCurrRcpTtlSlt;
	p_diLifterBtmPosInUM ACCESS p_MagRcpCurrRcpMag1Slt1Pos;
	p_diLifterCurrPosInUM ACCESS p_LifterBtmActualPos;
	p_bGdBrdIn ACCESS p_PshrConvGdBrd;
	p_bNxtLoadSeq ACCESS p_NtParamBffr1NxtLoadSeq;
//	p_bMagPresentSensor ACCESS p_DIMagPresentSen1;
	p_sCurrRcpNm ACCESS p_ProdRcpCurrRcp2Nm;
	p_sProgNm ACCESS p_NtParamBffr1ProgNm;
	p_bNtSettingsLoadDone ACCESS p_StartupNtSettingsLoadDone;
	p_bNtParamAutoRcpPrep ACCESS p_NtParamAutoRcpPrep ;
	p_bMcParamAutoRcpDis  ACCESS p_McParamAutoRcpDisable;

	//Siemens Req
	p_bOpsMagConvULRlsMagAllw ACCESS p_OpsMagConvUL1RlsMagAllw;
	p_eNtParamCustomerReq ACCESS p_NtParamCustomerReq;
	p_tyResponseFromMES ACCESS p_TagFromMesMagConv1;

	p_bNtParamAutoRcpF1ArbitraryType ACCESS p_NtParamAutoRcpF1ArbitraryType;
	(* Always Change If Project Change *)

END_ACTION
```

#### Act_InitLocal.st
```iecst
(** 2019-07-03 **)
ACTION Act_InitLocal:

	//Input Reference Link To Local Variable
	p_eAct ACCESS ADR(eAct);
	p_udiRstErr ACCESS ADR(udiRstErr);
	p_sFileName ACCESS ADR(sFileName);
	p_bManual ACCESS ADR(bManual);
	p_dtCurrDT ACCESS ADR(dtCurrDT);
	p_diMinSlt ACCESS ADR(diMinSlt);
	p_diMaxSlt ACCESS ADR(diMaxSlt);
	p_diPitch ACCESS ADR(diPitch);
	p_diSltCap ACCESS ADR(diSltCap);
	p_diBffrTtlSlt ACCESS ADR(diBffrTtlSlt);
	p_diCoolTm ACCESS ADR(diCoolTm);
	p_diSltToSltInUM ACCESS ADR(diSltToSltInUM);
	p_diLifterBtmPosInUM ACCESS ADR(diLifterBtmPosInUM);
	p_diLifterCurrPosInUM ACCESS ADR(diLifterCurrPosInUM);
	p_bAscending ACCESS ADR(bAscending);
	p_bFIFO ACCESS ADR(bFIFO);
	p_bGdBrdIn ACCESS ADR(bGdBrdIn);
	p_bGdBrdReq ACCESS ADR(bGdBrdReq);
	p_bNxtLoadSeq ACCESS ADR(bNxtLoadSeq);
	pa_bSkip ACCESS ADR(a_bSkip);
	p_diCoolFanOffDlyTm ACCESS ADR(diCoolFanOffDlyTm);
	p_bMagPresentSensor ACCESS ADR(bMagPresentSensor);
	p_bPrepCoolFan ACCESS ADR(bPrepCoolFan);
	p_bCoolFanTm ACCESS ADR(bCoolFanTm);
	p_tyBuffer ACCESS ADR(tyBuffer);
	p_tyDispBuffer ACCESS ADR(tyDispBuffer);
	p_tyBufferStat ACCESS ADR(tyBufferStat);
	p_sBffrNm ACCESS ADR(sBffrNm);
	p_sProdNm ACCESS ADR(sProdNm);
	p_sBarcode1 ACCESS ADR(sBarcode1);
	p_sBarcode2 ACCESS ADR(sBarcode2);
	p_sCurrRcpNm ACCESS ADR(sCurrRcpNm);
	p_sProgNm ACCESS ADR(sProgNm);
	p_bNtSettingsLoadDone ACCESS ADR(bNtSettingsLoadDone);

END_ACTION
```

#### Act_InputConfig.st
```iecst
(** 2019-04-26 **)
ACTION Act_InputConfig:

	(* Always Change If Project Change *)

	//Pass Data To Link
	tylocalBuffer.In.bLinkPresentSen1 := g_tyDInput.bMagPresentSen1;
	tylocalBuffer.In.bLinkPresentSen2 := g_tyDInput.bMagConvEntSen1;
	tylocalBuffer.In.diLinkSltToSltDist ACCESS p_MagRcpCurrRcpSltToSlt;
	tylocalBuffer.In.bLinkMcParamProdSelTopToBtm ACCESS p_ProdRcpCurrRcp2TopToBtm;
	tylocalBuffer.In.bLinkOpsTravLifULExitBrd ACCESS p_OpsTravLifULExitBrd;

	//Pass Data To Internal Use
	tylocalBuffer.In.udiRstErr := g_tyRstErr.bReset;
	tylocalBuffer.In.sFileName := g_tyNtParamCurr.sBffr1FileNm;
	tylocalBuffer.In.bManual := g_tyUIOut.bManualMod;
	tylocalBuffer.In.dtCurrDT := g_tyTime.dtCurrDT;

	tylocalBuffer.In.diBffrTtlSlt ACCESS p_MagRcpCurrRcpTtlSlt;
	tylocalBuffer.In.diLifterBtmPosInUM ACCESS p_MagRcpCurrRcpMag1Slt1Pos;
	tylocalBuffer.In.diLifterCurrPosInUM := g_tyLifterBtm.diActualPos;
	tylocalBuffer.In.bGdBrdIn  := g_tyPshrConv.bGdBrd;
	tylocalBuffer.In.bNxtLoadSeq := g_tyNtParamCurr.bBffr1NxtLoadSeq;
	tylocalBuffer.In.sCurrRcpNm ACCESS p_ProdRcpCurrRcp2Nm;
	tylocalBuffer.In.sProgNm := g_tyNtParamCurr.sBffr1ProgNm;
	tylocalBuffer.In.bNtParamAutoRcpPrep := g_tyNtParamCurr.bAutoRcpPrep ;
	tylocalBuffer.In.bMcParamAutoRcpDis  := g_tyMcParamCurr.bAutoRcpDisable;

	//Siemens Req
	tylocalBuffer.In.bOpsMagConvULRlsMagAllw := g_tyOpsMagConvUL1.bRlsMagAllw;
	tylocalBuffer.In.eNtParamCustomerReq := g_tyNtParamCurr.eCustomerReq;
	tylocalBuffer.In.tyResponseFromMES :=  g_tyAGV.tyTagFromMesMagCov1;
	(* Always Change If Project Change *)

	IF g_tyStartUp.bRun = TRUE THEN
		tylocalBuffer.In.eAct := g_tyStartUp.eBuffer1Act;
	ELSE
		IF tylocalBuffer.Out.eStatus = Idle THEN
			IF g_tyNtParamCurr.bProjLifterMagPlatform = FALSE THEN
				IF g_tyOpsMagConvUL1.eBufferAct <> BufferActIdle THEN
					tylocalBuffer.In.eAct := g_tyOpsMagConvUL1.eBufferAct;
				ELSIF g_tyUIOut.eBuffer1Act <> BufferActIdle THEN
					tylocalBuffer.In.eAct := g_tyUIOut.eBuffer1Act;
				ELSE
					tylocalBuffer.In.eAct := eAct;
				END_IF
			ELSE
				IF g_tyOpsLifMagULBufferAct1.eBufferAct <> BufferActIdle THEN
					tylocalBuffer.In.eAct := g_tyOpsLifMagULBufferAct1.eBufferAct;
				ELSE
					tylocalBuffer.In.eAct := g_tyUIOut.eBuffer1Act;
				END_IF
			END_IF
		END_IF
	END_IF

END_ACTION
```

#### Act_Link.st
```iecst
(** 2019-03-29 **)
ACTION Act_Link:
	IF g_tyNtParamCurr.bAutoRcpPrep AND NOT(g_tyMcParamCurr.bAutoRcpDisable) THEN
		tylocalBuffer.In.diMinSlt ACCESS g_tyAutoRcpMag1.diMinSlt;
		tylocalBuffer.In.diMaxSlt ACCESS g_tyAutoRcpMag1.diMaxSlt;
		tylocalBuffer.In.diPitch ACCESS g_tyAutoRcpMag1.diPitch;
	ELSE
		tylocalBuffer.In.diMinSlt ACCESS p_ProdRcpCurrRcp2MinSltValue;
		tylocalBuffer.In.diMaxSlt ACCESS p_ProdRcpCurrRcp2MaxSltValue;
		tylocalBuffer.In.diPitch ACCESS p_ProdRcpCurrRcp2Pitch;
	END_IF
	IF g_tyNtParamCurr.bProjLifterMagPlatform THEN
		tylocalBuffer.In.diSltToSltInUM ACCESS p_MagRcpCurrRcpSltToSlt;
	ELSE
		tylocalBuffer.In.diSltToSltInUM	:= tylocalBuffer.In.diLinkSltToSltDist * -1;
	END_IF

	tylocalBuffer.In.bAscending	:= NOT tylocalBuffer.In.bLinkMcParamProdSelTopToBtm;

	IF tylocalBuffer.In.bLinkOpsTravLifULExitBrd THEN
		tylocalBuffer.In.bMagPresentSensor := tylocalBuffer.In.bLinkPresentSen1; //present sensor only
	ELSE
		tylocalBuffer.In.bMagPresentSensor := tylocalBuffer.In.bLinkPresentSen1 OR tylocalBuffer.In.bLinkPresentSen2;
	END_IF

	//For MES Call Full
	IF tylocalBuffer.In.tyResponseFromMES.bTrigMagFull AND tylocalBuffer.In.bOpsMagConvULRlsMagAllw
		AND NOT(tylocalBuffer.Out.tyBufferStat.bBffrFull)  AND tylocalBuffer.In.eNtParamCustomerReq = Siemens THEN
		bMESTrigSetFull	:= TRUE;
	END_IF
	IF bMESTrigSetFull THEN
		tylocalBuffer.In.eAct	:= BufferActSetFull;
		IF tylocalBuffer.Out.eStat = BufferActSetFull AND tylocalBuffer.Out.eStatus = Done THEN
			tylocalBuffer.In.eAct	:= BufferActIdle;
			bMESTrigSetFull := FALSE;
		END_IF
	END_IF

END_ACTION
```

#### Act_LinkAction.st
```iecst
(** 2019-05-10 **)
ACTION Act_LinkAction:

	IF p_bLinkStartupRun = TRUE THEN
		p_eAct ACCESS p_StartupBuffer1Act;
	ELSE
		IF eStatus = Idle THEN
			IF p_bLinkProjLifterMagPlatform = FALSE THEN
				IF p_eLinkOpsMagConvULBufferAct <> BufferActIdle THEN
					p_eAct ACCESS p_OpsMagConvUL1BufferAct;
				ELSIF p_eLinkUIBufferAct <> BufferActIdle THEN
					p_eAct ACCESS p_UIBuffer1Act;
				ELSE
					p_eAct ACCESS ADR(eAct);
				END_IF
			ELSE
				IF p_eLinkOpsLifMagULBufferAct <> BufferActIdle THEN
					p_eAct ACCESS p_OpsLifMagULBufferAct1;
				ELSE
					p_eAct ACCESS p_UIBuffer1Act;
				END_IF
			END_IF
		END_IF
	END_IF

END_ACTION
```

#### Act_OutputConfig.st
```iecst
ACTION Act_OutputConfig:

	g_tyBuffer1 := tylocalBuffer.Out;

END_ACTION
```

#### Init.st
```iecst
(** 2019-06-07 **)
PROGRAM _INIT

	(* Always Change If Project Change *)

	//Pass Address To Global Address For External Use
	//Action, State & Status
	p_Buffer1Stat		:= ADR(eStat);
	p_Buffer1Status		:= ADR(eStatus);
	p_Buffer1StatTxt	:= ADR(sStatTxt);

	//Alarm
	p_Buffer1AlmData	:= ADR(tyAlmData);

	//Output
	p_Buffer1NxtLoadSlt				:= ADR(diNxtLoadSlt);
	p_Buffer1NxtUnloadSlt			:= ADR(diNxtUnloadSlt);
	p_Buffer1CoolBrdAny				:= ADR(diCoolBrdAny);
	p_Buffer1CoolBrdGd				:= ADR(diCoolBrdGd);
	p_Buffer1CoolBrdBad				:= ADR(diCoolBrdBad);
	p_Buffer1CoolNotRdy				:= ADR(bCoolNotRdy);
	p_Buffer1Bffr					:= ADR(tyBuffer);
	p_Buffer1DispBffr				:= ADR(tyDispBuffer);
	p_Buffer1BffrStat				:= ADR(tyBufferStat);
	p_Buffer1BrdUnloadStat			:= ADR(tyBoardUnloadStat);
	p_Buffer1FileNotFound			:= ADR(bFileNotFound);
	p_Buffer1CoolFanCtrl			:= ADR(bCoolFanCtrl);
	p_Buffer1MagPresent				:= ADR(bMagPresent);
	p_Buffer1MagPresentTm			:= ADR(dtMagPresentTm);
	p_Buffer1NewProduct				:= ADR(bNewProduct);
	p_Buffer1LastProductUnload		:= ADR(bLastProductUnload);
	p_Buffer1LastProductLeftInBffr	:= ADR(bLastProductLeftInBffr);
	p_Buffer1ParamDiff				:= ADR(bParamDiff);
	p_Buffer1MagRemoved				:= ADR(bMagRemoved);
	p_Buffer1FIFOOld				:= ADR(bFIFOOld);

	//Svy Hermes
	p_Buffer1SlotNo					:= ADR(diCurrSlt);
	(* Always Change If Project Change *)

END_PROGRAM
```

### Program Logical/Buffer/Buffer2 (IEC, version 1.00.0) - 1.00.0 - NtBuffer v5.00.0 , NtFileIO v5.00.0

#### Init.st - Change By Project
```iecst
(** 2019-06-07 **)
PROGRAM _INIT

	(* Always Change If Project Change *)

	//Pass Address To Global Address For External Use
	//Action, State & Status
	p_Buffer2Stat		:= ADR(eStat);
	p_Buffer2Status		:= ADR(eStatus);
	p_Buffer2StatTxt	:= ADR(sStatTxt);

	//Alarm
	p_Buffer2AlmData	:= ADR(tyAlmData);

	//Output
	p_Buffer2NxtLoadSlt				:= ADR(diNxtLoadSlt);
	p_Buffer2NxtUnloadSlt			:= ADR(diNxtUnloadSlt);
	p_Buffer2CoolBrdAny				:= ADR(diCoolBrdAny);
	p_Buffer2CoolBrdGd				:= ADR(diCoolBrdGd);
	p_Buffer2CoolBrdBad				:= ADR(diCoolBrdBad);
	p_Buffer2CoolNotRdy				:= ADR(bCoolNotRdy);
	p_Buffer2Bffr					:= ADR(tyBuffer);
	p_Buffer2DispBffr				:= ADR(tyDispBuffer);
	p_Buffer2BffrStat				:= ADR(tyBufferStat);
	p_Buffer2BrdUnloadStat			:= ADR(tyBoardUnloadStat);
	p_Buffer2FileNotFound			:= ADR(bFileNotFound);
	p_Buffer2CoolFanCtrl			:= ADR(bCoolFanCtrl);
	p_Buffer2MagPresent				:= ADR(bMagPresent);
	p_Buffer2MagPresentTm			:= ADR(dtMagPresentTm);
	p_Buffer2NewProduct				:= ADR(bNewProduct);
	p_Buffer2LastProductUnload		:= ADR(bLastProductUnload);
	p_Buffer2LastProductLeftInBffr	:= ADR(bLastProductLeftInBffr);
	p_Buffer2ParamDiff				:= ADR(bParamDiff);
	p_Buffer2MagRemoved				:= ADR(bMagRemoved);
	p_Buffer2FIFOOld				:= ADR(bFIFOOld);

	//Svy Hermes
	p_Buffer2SlotNo					:= ADR(diCurrSlt);
	(* Always Change If Project Change *)

END_PROGRAM
```

#### Act_InitGlobal.st - Change By Project
```iecst
(** 2019-04-26 **)
ACTION Act_InitGlobal:

	(* Always Change If Project Change *)

	//Pass Data To Link
	p_bLinkStartupRun ACCESS p_StartupRun;
	p_bLinkNtParamProjMagConvPrep ACCESS p_NtParamProjMag2ConvPrep;
//	p_eLinkOpsMagULBufferAct ACCESS p_OpsMagUL2BufferAct;
	p_eLinkOpsMagConvULBufferAct ACCESS p_OpsMagConvUL2BufferAct;
	p_eLinkUIBufferAct ACCESS p_UIBuffer2Act;
	p_bLinkProjLifterMagPlatform ACCESS p_NtParamProjLifterMagPlatform;
	p_eLinkOpsLifMagULBufferAct ACCESS p_OpsLifMagULBufferAct2;

	p_diLinkSltToSltDist ACCESS p_MagRcpCurrRcpSltToSlt;
	p_bLinkMcParamProdSelTopToBtm ACCESS p_ProdRcpCurrRcp2TopToBtm;
	p_bLinkPresentSen1 ACCESS p_DIMagPresentSen2;
	p_bLinkPresentSen2 ACCESS p_DIMagConvEntSen2;
	p_bLinkProjLifter2Prep ACCESS p_NtParamProjLifter2Prep;
	p_bLinkOpsTravLifULExitBrd ACCESS p_OpsTravLifULExitBrd;

	//Pass Data To Internal Use
	p_udiRstErr ACCESS p_RstErrReset;
	p_sFileName ACCESS p_NtParamBffr2FileNm;
	p_bManual ACCESS p_UIMnlMod;
	p_dtCurrDT ACCESS p_TimeCurrDT;

	p_diBffrTtlSlt ACCESS p_MagRcpCurrRcpTtlSlt;
	p_diLifterBtmPosInUM ACCESS p_MagRcpCurrRcpMag2Slt1Pos;
//	p_diLifterCurrPosInUM ACCESS p_LifterBtmActualPos;
	p_bGdBrdIn ACCESS p_PshrConvGdBrd;
	p_bNxtLoadSeq ACCESS p_NtParamBffr2NxtLoadSeq;
//	p_bMagPresentSensor ACCESS p_DIMagPresentSen2;
	p_sCurrRcpNm ACCESS p_ProdRcpCurrRcp2Nm;
	p_sProgNm ACCESS p_NtParamBffr2ProgNm;
	p_bNtSettingsLoadDone ACCESS p_StartupNtSettingsLoadDone;
	p_bNtParamAutoRcpPrep ACCESS p_NtParamAutoRcpPrep ;
	p_bMcParamAutoRcpDis  ACCESS p_McParamAutoRcpDisable;

	//Siemens Req
	p_bOpsMagConvULRlsMagAllw ACCESS p_OpsMagConvUL2RlsMagAllw;
	p_eNtParamCustomerReq ACCESS p_NtParamCustomerReq;
	p_tyResponseFromMES ACCESS p_TagFromMesMagConv2; //Siemens Req

	p_bNtParamAutoRcpF1ArbitraryType ACCESS p_NtParamAutoRcpF1ArbitraryType;
	(* Always Change If Project Change *)

END_ACTION
```

#### InputRef_Link.var - Change By Project
```iecst
(*2019-04-09*)
(**)
(*External*)
VAR
	p_bLinkStartupRun : REFERENCE TO BOOL;
	p_bLinkNtParamProjMagConvPrep : REFERENCE TO BOOL;
	p_eLinkOpsMagULBufferAct : REFERENCE TO eBufferAction;
	p_eLinkOpsMagConvULBufferAct : REFERENCE TO eBufferAction;
	p_eLinkUIBufferAct : REFERENCE TO eBufferAction;
END_VAR
(**)
VAR
	p_diLinkSltToSltDist : REFERENCE TO DINT;
	p_bLinkMcParamProdSelTopToBtm : REFERENCE TO BOOL;
	p_bLinkPresentSen1 : REFERENCE TO BOOL;
	p_bLinkPresentSen2 : REFERENCE TO BOOL;
	p_bLinkProjLifterMagPlatform : REFERENCE TO BOOL;
	p_eLinkOpsLifMagULBufferAct : REFERENCE TO eBufferAction;
	p_bLinkProjLifter2Prep : REFERENCE TO BOOL;
	p_bLinkOpsTravLifULExitBrd : REFERENCE TO BOOL;
END_VAR
```

#### Act_LinkAction.st - Change By Project
```iecst
(** 2019-05-10 **)
ACTION Act_LinkAction:

	IF p_bLinkStartupRun = TRUE THEN
		p_eAct ACCESS p_StartupBuffer2Act;
	ELSE
		IF eStatus = Idle THEN
			IF p_bLinkProjLifterMagPlatform = FALSE THEN
				IF p_eLinkOpsMagConvULBufferAct <> BufferActIdle THEN
					p_eAct ACCESS p_OpsMagConvUL2BufferAct;
				ELSIF p_eLinkUIBufferAct <> BufferActIdle THEN
					p_eAct ACCESS p_UIBuffer2Act;
				ELSE
					p_eAct ACCESS ADR(eAct);
				END_IF
			ELSE
				IF p_eLinkOpsLifMagULBufferAct <> BufferActIdle THEN
					p_eAct ACCESS p_OpsLifMagULBufferAct2;
				ELSE
					p_eAct ACCESS p_UIBuffer2Act;
				END_IF
			END_IF
		END_IF
	END_IF

END_ACTION
```

#### Act_Link.st - Change By Project
```iecst
(** 2019-03-29 **)
ACTION Act_Link:
	IF g_tyNtParamCurr.bAutoRcpPrep AND NOT(g_tyMcParamCurr.bAutoRcpDisable) THEN
		tylocalBuffer.In.diMinSlt ACCESS g_tyAutoRcpMag2.diMinSlt;
		tylocalBuffer.In.diMaxSlt ACCESS g_tyAutoRcpMag2.diMaxSlt;
		tylocalBuffer.In.diPitch ACCESS g_tyAutoRcpMag2.diPitch;
	ELSE
		tylocalBuffer.In.diMinSlt ACCESS p_ProdRcpCurrRcp2MinSltValue;
		tylocalBuffer.In.diMaxSlt ACCESS p_ProdRcpCurrRcp2MaxSltValue;
		tylocalBuffer.In.diPitch ACCESS p_ProdRcpCurrRcp2Pitch;
	END_IF
	IF g_tyNtParamCurr.bProjLifterMagPlatform THEN
		tylocalBuffer.In.diSltToSltInUM ACCESS p_MagRcpCurrRcpSltToSlt;
	ELSE
		tylocalBuffer.In.diSltToSltInUM	:= tylocalBuffer.In.diLinkSltToSltDist * -1;
	END_IF

	tylocalBuffer.In.bAscending	:= NOT tylocalBuffer.In.bLinkMcParamProdSelTopToBtm;

	IF tylocalBuffer.In.bLinkOpsTravLifULExitBrd THEN
		tylocalBuffer.In.bMagPresentSensor := tylocalBuffer.In.bLinkPresentSen1; //present sensor only
	ELSE
		tylocalBuffer.In.bMagPresentSensor := tylocalBuffer.In.bLinkPresentSen1 OR tylocalBuffer.In.bLinkPresentSen2;
	END_IF

	//For MES Call Full
	IF tylocalBuffer.In.tyResponseFromMES.bTrigMagFull AND tylocalBuffer.In.bOpsMagConvULRlsMagAllw
		AND NOT(tylocalBuffer.Out.tyBufferStat.bBffrFull)  AND tylocalBuffer.In.eNtParamCustomerReq = Siemens THEN
		bMESTrigSetFull	:= TRUE;
	END_IF
	IF bMESTrigSetFull THEN
		tylocalBuffer.In.eAct	:= BufferActSetFull;
		IF tylocalBuffer.Out.eStat = BufferActSetFull AND tylocalBuffer.Out.eStatus = Done THEN
			tylocalBuffer.In.eAct	:= BufferActIdle;
			bMESTrigSetFull := FALSE;
		END_IF
	END_IF

	IF g_tyNtParamCurr.bProjLifter2Prep THEN
		tylocalBuffer.In.diLifterCurrPosInUM := g_tyLifter2.diActualPos;
	ELSE
		tylocalBuffer.In.diLifterCurrPosInUM := g_tyLifterBtm.diActualPos;
	END_IF
END_ACTION
```

#### Cyclic.st - Do Not Change!!!
```iecst
(** 2019-03-29 **)
PROGRAM _CYCLIC

	IF bInitDone = FALSE THEN
		bInitDone	:= TRUE;

		Act_InitLocal;
		Act_InitGlobal;

	ELSIF bInitialDone = FALSE THEN
		IF p_bNtSettingsLoadDone = TRUE THEN
			bInitialDone	:= TRUE;

			Act_Initial;
		END_IF

	ELSE

		Act_Background;
		Act_RstErr;
		Act_LinkAction;
		Act_Action;
		Act_Link;
		Act_Main;
		Act_Alarm;

	END_IF

END_PROGRAM
```

#### Act_Initial.st - Do Not Change!!!
```iecst
(** 2019-04-26 **)
ACTION Act_Initial:

	//Initial
	sStatTxt	:= a_sStatText[eStat];

	fbDirCreate1.sDevice	:= 'F';
	fbDirCreate1.sDirName	:= 'User';
	fbDirCreate1(bEn := FALSE);

	fbDirCreate2.sDevice	:= 'User';
	fbDirCreate2.sDirName	:= 'Retain';
	fbDirCreate2(bEn := FALSE);

	fbFileRead1.sDevice			:= 'Retain';
	fbFileRead1.sFile			:= p_sFileName;
	fbFileRead1.udiOffset		:= 0;
	fbFileRead1.p_Dest			:= ADR(p_tyBuffer);
	fbFileRead1.udiLen			:= SIZEOF(p_tyBuffer);
	fbFileRead1(bEn := FALSE);

	fbFileWrite1.sDevice		:= 'Retain';
	fbFileWrite1.sFile			:= p_sFileName;
	fbFileWrite1.udiOffset		:= 0;
	fbFileWrite1.p_Src			:= ADR(p_tyBuffer);
	fbFileWrite1.udiLen			:= SIZEOF(p_tyBuffer);
	fbFileWrite1.udiOption		:= 0;
	fbFileWrite1(bEn := FALSE);

	fbCoolFanOffDlyTm.PT	:= DINT_TO_TIME(p_diCoolFanOffDlyTm);
	fbCoolFanOffDlyTm(IN := FALSE);

	fbCoolFanOffChkTm(IN := FALSE);
	fbMagAbsentTm(IN := FALSE);
	fbMagPresentTm(IN := FALSE);

END_ACTION
```

#### Act_Action.st - Do Not Change!!!
```iecst
(** 2019-03-25 **)
ACTION Act_Action:

	//Reset Error
	IF (eStatus = Error) AND bRstErr THEN
		p_eAct	:= BufferActIdle;
		eStat	:= BufferActIdle;
	END_IF

	//Set p_eAct
	IF eStatus = Idle OR eStatus = Busy OR eStatus = Done THEN
		eStat	:= p_eAct;
	END_IF

END_ACTION
```
